LIN {X 0.085,Y -554.089,Z 631.442,A 0.000,B 0.000,C 90.000,E1 115.540} C_DIS
LIN {X 0.039,Y -558.217,Z 631.438,A 0.000,B 0.000,C 90.000,E1 114.847} C_DIS
LIN {X 0.028,Y -561.886,Z 631.434,A 0.000,B 0.000,C 90.000,E1 114.155} C_DIS
LIN {X -0.047,Y -565.879,Z 631.430,A 0.000,B 0.000,C 90.000,E1 113.334} C_DIS
LIN {X 0.254,Y -570.586,Z 631.424,A 0.000,B 0.000,C 90.000,E1 112.206} C_DIS
LIN {X 0.040,Y -573.804,Z 631.419,A 0.000,B 0.000,C 90.000,E1 111.408} C_DIS
LIN {X 0.026,Y -575.811,Z 631.416,A 0.000,B 0.000,C 90.000,E1 110.865} C_DIS
LIN {X -0.133,Y -578.606,Z 631.411,A 0.000,B 0.000,C 90.000,E1 110.066} C_DIS
LIN {X -0.267,Y -581.153,Z 631.407,A 0.000,B 0.000,C 90.000,E1 109.268} C_DIS
LIN {X 0.171,Y -583.428,Z 631.402,A 0.000,B 0.000,C 90.000,E1 108.417} C_DIS
LIN {X -0.105,Y -585.449,Z 631.398,A 0.000,B 0.000,C 90.000,E1 107.638} C_DIS
LIN {X 0.203,Y -587.394,Z 631.393,A 0.000,B 0.000,C 90.000,E1 106.804} C_DIS
LIN {X 0.014,Y -591.886,Z 631.383,A 0.000,B 0.000,C 90.000,E1 104.954} C_DIS
LIN {X 0.067,Y -595.897,Z 631.374,A 0.000,B 0.000,C 90.000,E1 103.355} C_DIS
LIN {X -0.234,Y -599.246,Z 631.367,A 0.000,B 0.000,C 90.000,E1 102.063} C_DIS
LIN {X 0.103,Y -602.617,Z 631.360,A 0.000,B 0.000,C 90.000,E1 100.715} C_DIS
LIN {X -0.213,Y -605.836,Z 631.352,A 0.000,B 0.000,C 90.000,E1 99.434} C_DIS
LIN {X 0.029,Y -608.811,Z 631.345,A 0.000,B 0.000,C 90.000,E1 98.106} C_DIS
LIN {X -0.005,Y -611.109,Z 631.339,A 0.000,B 0.000,C 90.000,E1 97.068} C_DIS
LIN {X -0.273,Y -613.680,Z 631.332,A 0.000,B 0.000,C 90.000,E1 95.796} C_DIS
LIN {X 0.024,Y -615.053,Z 631.328,A 0.000,B 0.000,C 90.000,E1 94.992} C_DIS
LIN {X -0.248,Y -617.171,Z 631.321,A 0.000,B 0.000,C 90.000,E1 93.726} C_DIS
LIN {X -0.222,Y -618.720,Z 631.315,A 0.000,B 0.000,C 90.000,E1 92.694} C_DIS
LIN {X 0.139,Y -620.287,Z 631.308,A 0.000,B 0.000,C 90.000,E1 91.375} C_DIS
LIN {X -0.136,Y -621.077,Z 631.303,A 0.000,B 0.000,C 90.000,E1 90.630} C_DIS
LIN {X -0.075,Y -621.849,Z 631.298,A 0.000,B 0.000,C 90.000,E1 89.599} C_DIS
LIN {X -0.301,Y -622.416,Z 631.291,A 0.000,B 0.000,C 90.000,E1 88.339} C_DIS
LIN {X -0.208,Y -622.576,Z 631.285,A 0.000,B 0.000,C 90.000,E1 87.306} C_DIS
LIN {X 0.211,Y -622.380,Z 631.278,A 0.000,B 0.000,C 90.000,E1 85.988} C_DIS
LIN {X -0.270,Y -621.941,Z 631.272,A 0.000,B 0.000,C 90.000,E1 85.008} C_DIS
LIN {X 0.183,Y -621.213,Z 631.265,A 0.000,B 0.000,C 90.000,E1 83.685} C_DIS
LIN {X 0.073,Y -620.135,Z 631.258,A 0.000,B 0.000,C 90.000,E1 82.413} C_DIS
LIN {X -0.104,Y -619.289,Z 631.254,A 0.000,B 0.000,C 90.000,E1 81.659} C_DIS
LIN {X -0.012,Y -617.891,Z 631.248,A 0.000,B 0.000,C 90.000,E1 80.622} C_DIS
LIN {X 0.151,Y -616.382,Z 631.242,A 0.000,B 0.000,C 90.000,E1 79.577} C_DIS
LIN {X 0.168,Y -614.185,Z 631.235,A 0.000,B 0.000,C 90.000,E1 78.285} C_DIS
LIN {X -0.194,Y -612.299,Z 631.229,A 0.000,B 0.000,C 90.000,E1 77.285} C_DIS
LIN {X -0.233,Y -609.621,Z 631.222,A 0.000,B 0.000,C 90.000,E1 75.992} C_DIS
LIN {X -0.071,Y -607.405,Z 631.216,A 0.000,B 0.000,C 90.000,E1 74.936} C_DIS
LIN {X 0.112,Y -604.394,Z 631.209,A 0.000,B 0.000,C 90.000,E1 73.614} C_DIS
LIN {X -0.222,Y -601.806,Z 631.203,A 0.000,B 0.000,C 90.000,E1 72.598} C_DIS
LIN {X 0.262,Y -599.743,Z 631.199,A 0.000,B 0.000,C 90.000,E1 71.764} C_DIS
LIN {X -0.126,Y -598.233,Z 631.196,A 0.000,B 0.000,C 90.000,E1 71.275} C_DIS
LIN {X -0.057,Y -595.727,Z 631.192,A 0.000,B 0.000,C 90.000,E1 70.477} C_DIS
LIN {X 0.096,Y -594.011,Z 631.189,A 0.000,B 0.000,C 90.000,E1 69.934} C_DIS
LIN {X -0.197,Y -590.097,Z 631.183,A 0.000,B 0.000,C 90.000,E1 68.901} C_DIS
LIN {X -0.210,Y -586.932,Z 631.178,A 0.000,B 0.000,C 90.000,E1 68.103} C_DIS
LIN {X -0.034,Y -583.567,Z 631.174,A 0.000,B 0.000,C 90.000,E1 67.283} C_DIS
LIN {X -0.187,Y -579.320,Z 631.169,A 0.000,B 0.000,C 90.000,E1 66.357} C_DIS
LIN {X -0.091,Y -575.356,Z 631.164,A 0.000,B 0.000,C 90.000,E1 65.537} C_DIS
LIN {X 0.139,Y -572.004,Z 631.160,A 0.000,B 0.000,C 90.000,E1 64.845} C_DIS
LIN {X 0.152,Y -567.287,Z 631.156,A 0.000,B 0.000,C 90.000,E1 64.024} C_DIS
LIN {X -0.069,Y -564.081,Z 631.153,A 0.000,B 0.000,C 90.000,E1 63.512} C_DIS
LIN {X -0.045,Y -559.282,Z 631.149,A 0.000,B 0.000,C 90.000,E1 62.820} C_DIS
LIN {X -0.196,Y -555.143,Z 631.146,A 0.000,B 0.000,C 90.000,E1 62.281} C_DIS
LIN {X -0.143,Y -550.650,Z 631.143,A 0.000,B 0.000,C 90.000,E1 61.719} C_DIS
LIN {X -0.182,Y -545.605,Z 631.140,A 0.000,B 0.000,C 90.000,E1 61.179} C_DIS
LIN {X -0.231,Y -541.679,Z 631.138,A 0.000,B 0.000,C 90.000,E1 60.795} C_DIS
LIN {X -0.230,Y -536.321,Z 631.135,A 0.000,B 0.000,C 90.000,E1 60.333} C_DIS
LIN {X -0.030,Y -530.617,Z 631.133,A 0.000,B 0.000,C 90.000,E1 59.871} C_DIS
LIN {X -0.118,Y -524.164,Z 631.130,A 0.000,B 0.000,C 90.000,E1 59.459} C_DIS
LIN {X 0.119,Y -515.999,Z 631.128,A 0.000,B 0.000,C 90.000,E1 58.948} C_DIS
LIN {X 0.131,Y -510.785,Z 631.126,A 0.000,B 0.000,C 90.000,E1 58.663} C_DIS
LIN {X -0.016,Y -503.911,Z 631.124,A 0.000,B 0.000,C 90.000,E1 58.329} C_DIS
LIN {X -0.137,Y -488.724,Z 631.120,A 0.000,B 0.000,C 90.000,E1 57.582} C_DIS
LIN {X -0.265,Y -467.090,Z 631.114,A 0.000,B 0.000,C 90.000,E1 56.501} C_DIS
LIN {X 0.064,Y -445.248,Z 631.107,A 0.000,B 0.000,C 90.000,E1 55.308} C_DIS
LIN {X -0.003,Y -440.385,Z 631.106,A 0.000,B 0.000,C 90.000,E1 55.055} C_DIS
LIN {X -0.047,Y -440.315,Z 631.106,A 0.000,B 0.000,C 90.000,E1 55.055} C_DIS
LIN {X -0.113,Y -431.751,Z 631.083,A 0.000,B 0.000,C 90.000,E1 50.964} C_DIS
LIN {X 0.067,Y -430.164,Z 631.079,A 0.000,B 0.000,C 90.000,E1 50.275} C_DIS
LIN {X -0.052,Y -425.382,Z 631.068,A 0.000,B 0.000,C 90.000,E1 48.243} C_DIS
LIN {X -0.081,Y -425.960,Z 631.061,A 0.000,B 0.000,C 90.000,E1 46.944} C_DIS
LIN {X 0.079,Y -426.371,Z 631.051,A 0.000,B 0.000,C 90.000,E1 45.243} C_DIS
LIN {X -0.214,Y -427.010,Z 631.038,A 0.000,B 0.000,C 90.000,E1 42.933} C_DIS
LIN {X 0.135,Y -427.902,Z 631.025,A 0.000,B 0.000,C 90.000,E1 40.539} C_DIS
LIN {X -0.059,Y -428.921,Z 631.012,A 0.000,B 0.000,C 90.000,E1 38.222} C_DIS
LIN {X -0.065,Y -429.888,Z 631.001,A 0.000,B 0.000,C 90.000,E1 36.217} C_DIS
LIN {X 0.053,Y -430.598,Z 630.992,A 0.000,B 0.000,C 90.000,E1 34.532} C_DIS
LIN {X 0.054,Y -430.923,Z 630.988,A 0.000,B 0.000,C 90.000,E1 33.865} C_DIS
LIN {X -0.039,Y -431.638,Z 630.977,A 0.000,B 0.000,C 90.000,E1 31.878} C_DIS
LIN {X 0.030,Y -432.485,Z 630.964,A 0.000,B 0.000,C 90.000,E1 29.539} C_DIS
LIN {X 0.267,Y -433.344,Z 630.953,A 0.000,B 0.000,C 90.000,E1 27.513} C_DIS
LIN {X 0.133,Y -434.356,Z 630.940,A 0.000,B 0.000,C 90.000,E1 25.207} C_DIS
LIN {X 0.057,Y -435.441,Z 630.927,A 0.000,B 0.000,C 90.000,E1 22.898} C_DIS
LIN {X 0.182,Y -436.359,Z 630.918,A 0.000,B 0.000,C 90.000,E1 21.227} C_DIS
LIN {X -0.077,Y -437.108,Z 630.911,A 0.000,B 0.000,C 90.000,E1 19.939} C_DIS
LIN {X 0.026,Y -438.151,Z 630.900,A 0.000,B 0.000,C 90.000,E1 17.946} C_DIS
LIN {X 0.025,Y -439.291,Z 630.889,A 0.000,B 0.000,C 90.000,E1 15.969} C_DIS
LIN {X -0.100,Y -440.959,Z 630.874,A 0.000,B 0.000,C 90.000,E1 13.355} C_DIS
LIN {X -0.207,Y -442.712,Z 630.861,A 0.000,B 0.000,C 90.000,E1 11.074} C_DIS
LIN {X -0.175,Y -444.938,Z 630.847,A 0.000,B 0.000,C 90.000,E1 8.454} C_DIS
LIN {X -0.071,Y -446.894,Z 630.836,A 0.000,B 0.000,C 90.000,E1 6.486} C_DIS
LIN {X -0.151,Y -449.638,Z 630.822,A 0.000,B 0.000,C 90.000,E1 3.898} C_DIS
LIN {X 0.198,Y -451.560,Z 630.813,A 0.000,B 0.000,C 90.000,E1 2.236} C_DIS
LIN {X -0.106,Y -455.171,Z 630.797,A 0.000,B 0.000,C 90.000,E1 359.484} C_DIS
LIN {X -0.178,Y -458.582,Z 630.785,A 0.000,B 0.000,C 90.000,E1 357.249} C_DIS
LIN {X -0.107,Y -462.241,Z 630.772,A 0.000,B 0.000,C 90.000,E1 355.008} C_DIS
LIN {X 0.109,Y -466.017,Z 630.760,A 0.000,B 0.000,C 90.000,E1 352.761} C_DIS
LIN {X -0.192,Y -469.281,Z 630.749,A 0.000,B 0.000,C 90.000,E1 350.905} C_DIS
LIN {X -0.249,Y -471.967,Z 630.741,A 0.000,B 0.000,C 90.000,E1 349.342} C_DIS
LIN {X 0.053,Y -475.727,Z 630.729,A 0.000,B 0.000,C 90.000,E1 347.117} C_DIS
LIN {X 0.098,Y -479.596,Z 630.716,A 0.000,B 0.000,C 90.000,E1 344.936} C_DIS
LIN {X 0.040,Y -483.665,Z 630.704,A 0.000,B 0.000,C 90.000,E1 342.779} C_DIS
LIN {X -0.241,Y -486.681,Z 630.696,A 0.000,B 0.000,C 90.000,E1 341.275} C_DIS
LIN {X 0.149,Y -489.655,Z 630.687,A 0.000,B 0.000,C 90.000,E1 339.699} C_DIS
LIN {X -0.107,Y -493.167,Z 630.677,A 0.000,B 0.000,C 90.000,E1 337.901} C_DIS
LIN {X 0.025,Y -494.765,Z 630.672,A 0.000,B 0.000,C 90.000,E1 336.975} C_DIS
LIN {X -0.180,Y -497.255,Z 630.664,A 0.000,B 0.000,C 90.000,E1 335.485} C_DIS
LIN {X 0.076,Y -499.568,Z 630.655,A 0.000,B 0.000,C 90.000,E1 333.948} C_DIS
LIN {X 0.002,Y -502.293,Z 630.645,A 0.000,B 0.000,C 90.000,E1 332.153} C_DIS
LIN {X 0.149,Y -506.008,Z 630.632,A 0.000,B 0.000,C 90.000,E1 329.744} C_DIS
LIN {X 0.148,Y -509.819,Z 630.620,A 0.000,B 0.000,C 90.000,E1 327.661} C_DIS
LIN {X -0.162,Y -513.440,Z 630.612,A 0.000,B 0.000,C 90.000,E1 326.215} C_DIS
LIN {X 0.103,Y -515.315,Z 630.609,A 0.000,B 0.000,C 90.000,E1 325.595} C_DIS
LIN {X 0.028,Y -516.613,Z 630.607,A 0.000,B 0.000,C 90.000,E1 325.308} C_DIS
LIN {X -0.028,Y -518.300,Z 630.605,A 0.000,B 0.000,C 90.000,E1 324.975} C_DIS
LIN {X 0.088,Y -519.185,Z 630.605,A 0.000,B 0.000,C 90.000,E1 324.815} C_DIS
LIN {X -0.264,Y -520.383,Z 630.604,A 0.000,B 0.000,C 90.000,E1 324.689} C_DIS
LIN {X 0.103,Y -522.215,Z 630.602,A 0.000,B 0.000,C 90.000,E1 324.356} C_DIS
LIN {X -0.089,Y -526.231,Z 630.599,A 0.000,B 0.000,C 90.000,E1 323.909} C_DIS
LIN {X 0.108,Y -531.100,Z 630.597,A 0.000,B 0.000,C 90.000,E1 323.417} C_DIS
LIN {X -0.048,Y -534.048,Z 630.595,A 0.000,B 0.000,C 90.000,E1 323.176} C_DIS
LIN {X -0.132,Y -540.909,Z 630.592,A 0.000,B 0.000,C 90.000,E1 322.637} C_DIS
LIN {X -0.285,Y -550.938,Z 630.588,A 0.000,B 0.000,C 90.000,E1 321.823} C_DIS
LIN {X 0.137,Y -563.763,Z 630.582,A 0.000,B 0.000,C 90.000,E1 320.723} C_DIS
LIN {X -0.050,Y -572.217,Z 630.578,A 0.000,B 0.000,C 90.000,E1 320.033} C_DIS
LIN {X -0.220,Y -581.991,Z 630.573,A 0.000,B 0.000,C 90.000,E1 319.218} C_DIS
LIN {X -0.098,Y -590.110,Z 630.569,A 0.000,B 0.000,C 90.000,E1 318.485} C_DIS
LIN {X 0.000,Y -597.970,Z 630.565,A 0.000,B 0.000,C 90.000,E1 317.757} C_DIS
LIN {X -0.241,Y -602.878,Z 630.563,A 0.000,B 0.000,C 90.000,E1 317.310} C_DIS
LIN {X 0.060,Y -605.489,Z 630.561,A 0.000,B 0.000,C 90.000,E1 317.025} C_DIS
LIN {X 0.076,Y -610.159,Z 630.559,A 0.000,B 0.000,C 90.000,E1 316.539} C_DIS
LIN {X 0.043,Y -614.632,Z 630.556,A 0.000,B 0.000,C 90.000,E1 316.053} C_DIS
LIN {X -0.024,Y -618.922,Z 630.553,A 0.000,B 0.000,C 90.000,E1 315.567} C_DIS
LIN {X -0.329,Y -623.212,Z 630.550,A 0.000,B 0.000,C 90.000,E1 315.081} C_DIS
LIN {X -0.351,Y -630.233,Z 630.545,A 0.000,B 0.000,C 90.000,E1 314.190} C_DIS
LIN {X 0.165,Y -636.856,Z 630.540,A 0.000,B 0.000,C 90.000,E1 313.257} C_DIS
LIN {X 0.009,Y -642.290,Z 630.536,A 0.000,B 0.000,C 90.000,E1 312.528} C_DIS
LIN {X -0.239,Y -648.488,Z 630.531,A 0.000,B 0.000,C 90.000,E1 311.676} C_DIS
LIN {X 0.072,Y -654.390,Z 630.527,A 0.000,B 0.000,C 90.000,E1 310.782} C_DIS
LIN {X -0.005,Y -658.239,Z 630.523,A 0.000,B 0.000,C 90.000,E1 310.172} C_DIS
LIN {X -0.080,Y -661.081,Z 630.521,A 0.000,B 0.000,C 90.000,E1 309.688} C_DIS
LIN {X -0.018,Y -664.314,Z 630.517,A 0.000,B 0.000,C 90.000,E1 309.072} C_DIS
LIN {X -0.064,Y -666.726,Z 630.514,A 0.000,B 0.000,C 90.000,E1 308.588} C_DIS
LIN {X 0.093,Y -671.048,Z 630.509,A 0.000,B 0.000,C 90.000,E1 307.604} C_DIS
LIN {X 0.190,Y -673.983,Z 630.505,A 0.000,B 0.000,C 90.000,E1 306.870} C_DIS
LIN {X -0.088,Y -676.736,Z 630.501,A 0.000,B 0.000,C 90.000,E1 306.171} C_DIS
LIN {X 0.215,Y -680.835,Z 630.494,A 0.000,B 0.000,C 90.000,E1 304.945} C_DIS
LIN {X 0.181,Y -683.858,Z 630.489,A 0.000,B 0.000,C 90.000,E1 303.992} C_DIS
LIN {X -0.005,Y -686.037,Z 630.485,A 0.000,B 0.000,C 90.000,E1 303.293} C_DIS
LIN {X 0.246,Y -689.601,Z 630.478,A 0.000,B 0.000,C 90.000,E1 302.084} C_DIS
LIN {X 0.330,Y -692.272,Z 630.473,A 0.000,B 0.000,C 90.000,E1 301.131} C_DIS
LIN {X -0.267,Y -695.505,Z 630.467,A 0.000,B 0.000,C 90.000,E1 300.001} C_DIS
LIN {X 0.051,Y -698.955,Z 630.459,A 0.000,B 0.000,C 90.000,E1 298.565} C_DIS
LIN {X -0.111,Y -701.035,Z 630.454,A 0.000,B 0.000,C 90.000,E1 297.641} C_DIS
LIN {X 0.087,Y -702.418,Z 630.450,A 0.000,B 0.000,C 90.000,E1 296.924} C_DIS
LIN {X -0.018,Y -703.452,Z 630.446,A 0.000,B 0.000,C 90.000,E1 296.232} C_DIS
LIN {X -0.085,Y -703.687,Z 630.443,A 0.000,B 0.000,C 90.000,E1 295.771} C_DIS
LIN {X -0.107,Y -703.580,Z 630.442,A 0.000,B 0.000,C 90.000,E1 295.540} C_DIS
LIN {X -0.176,Y -702.515,Z 630.439,A 0.000,B 0.000,C 90.000,E1 295.079} C_DIS
LIN {X 0.104,Y -701.665,Z 630.438,A 0.000,B 0.000,C 90.000,E1 294.823} C_DIS
LIN {X 0.225,Y -699.045,Z 630.436,A 0.000,B 0.000,C 90.000,E1 294.463} C_DIS
LIN {X -0.143,Y -697.041,Z 630.435,A 0.000,B 0.000,C 90.000,E1 294.259} C_DIS
LIN {X -0.012,Y -695.571,Z 630.434,A 0.000,B 0.000,C 90.000,E1 294.131} C_DIS
LIN {X -0.023,Y -693.395,Z 630.434,A 0.000,B 0.000,C 90.000,E1 294.027} C_DIS
LIN {X 0.255,Y -686.989,Z 630.432,A 0.000,B 0.000,C 90.000,E1 293.770} C_DIS
LIN {X -0.216,Y -683.102,Z 630.432,A 0.000,B 0.000,C 90.000,E1 293.695} C_DIS
LIN {X -0.155,Y -680.635,Z 630.431,A 0.000,B 0.000,C 90.000,E1 293.643} C_DIS
LIN {X 0.228,Y -674.010,Z 630.431,A 0.000,B 0.000,C 90.000,E1 293.515} C_DIS
LIN {X -0.254,Y -664.941,Z 630.430,A 0.000,B 0.000,C 90.000,E1 293.462} C_DIS
LIN {X -0.082,Y -651.280,Z 630.429,A 0.000,B 0.000,C 90.000,E1 293.259} C_DIS
LIN {X -0.303,Y -639.642,Z 630.428,A 0.000,B 0.000,C 90.000,E1 293.078} C_DIS
LIN {X -0.087,Y -628.867,Z 630.427,A 0.000,B 0.000,C 90.000,E1 292.823} C_DIS
LIN {X -0.031,Y -615.450,Z 630.425,A 0.000,B 0.000,C 90.000,E1 292.461} C_DIS
LIN {X -0.061,Y -594.878,Z 630.421,A 0.000,B 0.000,C 90.000,E1 291.844} C_DIS
LIN {X -0.126,Y -579.185,Z 630.419,A 0.000,B 0.000,C 90.000,E1 291.354} C_DIS
LIN {X -0.041,Y -570.243,Z 630.417,A 0.000,B 0.000,C 90.000,E1 291.099} C_DIS
LIN {X -0.246,Y -563.976,Z 630.416,A 0.000,B 0.000,C 90.000,E1 290.918} C_DIS
LIN {X -0.301,Y -559.805,Z 630.415,A 0.000,B 0.000,C 90.000,E1 290.737} C_DIS
LIN {X 0.159,Y -558.684,Z 630.415,A 0.000,B 0.000,C 90.000,E1 290.610} C_DIS
LIN {X -0.035,Y -556.909,Z 630.414,A 0.000,B 0.000,C 90.000,E1 290.482} C_DIS
LIN {X -0.070,Y -556.884,Z 630.414,A 0.000,B 0.000,C 90.000,E1 290.482} C_DIS
LIN {X 0.037,Y -556.255,Z 630.413,A 0.000,B 0.000,C 90.000,E1 290.248} C_DIS
LIN {X 0.215,Y -555.883,Z 630.410,A 0.000,B 0.000,C 90.000,E1 289.812} C_DIS
LIN {X -0.241,Y -556.063,Z 630.406,A 0.000,B 0.000,C 90.000,E1 289.033} C_DIS
LIN {X -0.208,Y -556.015,Z 630.398,A 0.000,B 0.000,C 90.000,E1 287.638} C_DIS
LIN {X 0.063,Y -555.727,Z 630.392,A 0.000,B 0.000,C 90.000,E1 286.496} C_DIS
LIN {X 0.173,Y -555.389,Z 630.386,A 0.000,B 0.000,C 90.000,E1 285.371} C_DIS
LIN {X -0.130,Y -554.702,Z 630.378,A 0.000,B 0.000,C 90.000,E1 284.008} C_DIS
LIN {X 0.216,Y -553.824,Z 630.369,A 0.000,B 0.000,C 90.000,E1 282.299} C_DIS
LIN {X -0.246,Y -553.157,Z 630.361,A 0.000,B 0.000,C 90.000,E1 280.950} C_DIS
LIN {X -0.162,Y -552.433,Z 630.351,A 0.000,B 0.000,C 90.000,E1 279.265} C_DIS
LIN {X -0.174,Y -551.722,Z 630.342,A 0.000,B 0.000,C 90.000,E1 277.587} C_DIS
LIN {X -0.161,Y -550.947,Z 630.331,A 0.000,B 0.000,C 90.000,E1 275.625} C_DIS
LIN {X -0.223,Y -550.382,Z 630.320,A 0.000,B 0.000,C 90.000,E1 273.669} C_DIS
LIN {X 0.130,Y -549.922,Z 630.311,A 0.000,B 0.000,C 90.000,E1 271.949} C_DIS
LIN {X -0.130,Y -549.551,Z 630.303,A 0.000,B 0.000,C 90.000,E1 270.573} C_DIS
LIN {X 0.087,Y -549.082,Z 630.297,A 0.000,B 0.000,C 90.000,E1 269.427} C_DIS
LIN {X -0.189,Y -548.444,Z 630.289,A 0.000,B 0.000,C 90.000,E1 268.051} C_DIS
LIN {X 0.076,Y -547.871,Z 630.281,A 0.000,B 0.000,C 90.000,E1 266.617} C_DIS
LIN {X -0.228,Y -547.096,Z 630.273,A 0.000,B 0.000,C 90.000,E1 265.241} C_DIS
LIN {X 0.199,Y -545.764,Z 630.263,A 0.000,B 0.000,C 90.000,E1 263.223} C_DIS
LIN {X -0.147,Y -545.026,Z 630.258,A 0.000,B 0.000,C 90.000,E1 262.413} C_DIS
LIN {X 0.127,Y -543.834,Z 630.252,A 0.000,B 0.000,C 90.000,E1 261.254} C_DIS
LIN {X 0.075,Y -541.448,Z 630.239,A 0.000,B 0.000,C 90.000,E1 258.993} C_DIS
LIN {X 0.001,Y -539.980,Z 630.229,A 0.000,B 0.000,C 90.000,E1 257.297} C_DIS
LIN {X 0.012,Y -538.583,Z 630.220,A 0.000,B 0.000,C 90.000,E1 255.589} C_DIS
LIN {X 0.016,Y -537.544,Z 630.214,A 0.000,B 0.000,C 90.000,E1 254.448} C_DIS
LIN {X 0.115,Y -535.708,Z 630.204,A 0.000,B 0.000,C 90.000,E1 252.725} C_DIS
LIN {X -0.189,Y -534.014,Z 630.195,A 0.000,B 0.000,C 90.000,E1 251.040} C_DIS
LIN {X -0.269,Y -533.017,Z 630.190,A 0.000,B 0.000,C 90.000,E1 250.188} C_DIS
LIN {X -0.164,Y -531.434,Z 630.183,A 0.000,B 0.000,C 90.000,E1 249.028} C_DIS
LIN {X 0.111,Y -529.754,Z 630.177,A 0.000,B 0.000,C 90.000,E1 247.847} C_DIS
LIN {X -0.121,Y -527.856,Z 630.171,A 0.000,B 0.000,C 90.000,E1 246.719} C_DIS
LIN {X 0.105,Y -525.750,Z 630.164,A 0.000,B 0.000,C 90.000,E1 245.537} C_DIS
LIN {X 0.127,Y -524.095,Z 630.159,A 0.000,B 0.000,C 90.000,E1 244.665} C_DIS
LIN {X 0.180,Y -520.981,Z 630.151,A 0.000,B 0.000,C 90.000,E1 243.204} C_DIS
LIN {X 0.071,Y -517.162,Z 630.142,A 0.000,B 0.000,C 90.000,E1 241.463} C_DIS
LIN {X 0.115,Y -514.546,Z 630.135,A 0.000,B 0.000,C 90.000,E1 240.284} C_DIS
LIN {X 0.030,Y -512.489,Z 630.130,A 0.000,B 0.000,C 90.000,E1 239.410} C_DIS
LIN {X 0.170,Y -508.945,Z 630.122,A 0.000,B 0.000,C 90.000,E1 237.916} C_DIS
LIN {X 0.246,Y -505.244,Z 630.114,A 0.000,B 0.000,C 90.000,E1 236.421} C_DIS
LIN {X -0.056,Y -502.256,Z 630.107,A 0.000,B 0.000,C 90.000,E1 235.261} C_DIS
LIN {X -0.118,Y -499.092,Z 630.100,A 0.000,B 0.000,C 90.000,E1 234.069} C_DIS
LIN {X 0.056,Y -492.078,Z 630.085,A 0.000,B 0.000,C 90.000,E1 231.331} C_DIS
LIN {X -0.098,Y -488.282,Z 630.077,A 0.000,B 0.000,C 90.000,E1 229.828} C_DIS
LIN {X 0.004,Y -484.582,Z 630.068,A 0.000,B 0.000,C 90.000,E1 228.286} C_DIS
LIN {X -0.162,Y -480.044,Z 630.058,A 0.000,B 0.000,C 90.000,E1 226.458} C_DIS
LIN {X -0.018,Y -474.760,Z 630.046,A 0.000,B 0.000,C 90.000,E1 224.271} C_DIS
LIN {X 0.235,Y -470.463,Z 630.036,A 0.000,B 0.000,C 90.000,E1 222.366} C_DIS
LIN {X -0.005,Y -467.058,Z 630.027,A 0.000,B 0.000,C 90.000,E1 220.825} C_DIS
LIN {X -0.254,Y -463.651,Z 630.018,A 0.000,B 0.000,C 90.000,E1 219.277} C_DIS
LIN {X -0.171,Y -459.645,Z 630.008,A 0.000,B 0.000,C 90.000,E1 217.363} C_DIS
LIN {X 0.000,Y -455.235,Z 629.995,A 0.000,B 0.000,C 90.000,E1 215.105} C_DIS
LIN {X 0.081,Y -451.710,Z 629.984,A 0.000,B 0.000,C 90.000,E1 213.166} C_DIS
LIN {X -0.093,Y -447.591,Z 629.972,A 0.000,B 0.000,C 90.000,E1 210.924} C_DIS
LIN {X 0.096,Y -444.173,Z 629.961,A 0.000,B 0.000,C 90.000,E1 208.949} C_DIS
LIN {X -0.009,Y -440.665,Z 629.950,A 0.000,B 0.000,C 90.000,E1 207.001} C_DIS
LIN {X 0.137,Y -438.382,Z 629.943,A 0.000,B 0.000,C 90.000,E1 205.668} C_DIS
LIN {X 0.084,Y -434.772,Z 629.932,A 0.000,B 0.000,C 90.000,E1 203.695} C_DIS
LIN {X 0.175,Y -431.877,Z 629.923,A 0.000,B 0.000,C 90.000,E1 202.025} C_DIS
LIN {X 0.075,Y -427.901,Z 629.910,A 0.000,B 0.000,C 90.000,E1 199.704} C_DIS
LIN {X 0.135,Y -424.096,Z 629.897,A 0.000,B 0.000,C 90.000,E1 197.347} C_DIS
LIN {X 0.126,Y -421.492,Z 629.887,A 0.000,B 0.000,C 90.000,E1 195.662} C_DIS
LIN {X -0.165,Y -418.953,Z 629.878,A 0.000,B 0.000,C 90.000,E1 194.008} C_DIS
LIN {X -0.042,Y -415.754,Z 629.866,A 0.000,B 0.000,C 90.000,E1 191.951} C_DIS
LIN {X -0.005,Y -411.834,Z 629.851,A 0.000,B 0.000,C 90.000,E1 189.208} C_DIS
LIN {X 0.101,Y -409.424,Z 629.842,A 0.000,B 0.000,C 90.000,E1 187.473} C_DIS
LIN {X 0.142,Y -405.681,Z 629.826,A 0.000,B 0.000,C 90.000,E1 184.702} C_DIS
LIN {X -0.067,Y -402.437,Z 629.811,A 0.000,B 0.000,C 90.000,E1 181.949} C_DIS
LIN {X -0.026,Y -399.449,Z 629.793,A 0.000,B 0.000,C 90.000,E1 178.797} C_DIS
LIN {X 0.144,Y -396.808,Z 629.768,A 0.000,B 0.000,C 90.000,E1 174.204} C_DIS
LIN {X -0.189,Y -396.039,Z 629.752,A 0.000,B 0.000,C 90.000,E1 171.432} C_DIS
LIN {X 0.064,Y -395.686,Z 629.739,A 0.000,B 0.000,C 90.000,E1 168.926} C_DIS
LIN {X -0.032,Y -395.779,Z 629.723,A 0.000,B 0.000,C 90.000,E1 166.117} C_DIS
LIN {X 0.131,Y -396.029,Z 629.711,A 0.000,B 0.000,C 90.000,E1 163.976} C_DIS
LIN {X 0.107,Y -396.478,Z 629.697,A 0.000,B 0.000,C 90.000,E1 161.511} C_DIS
LIN {X -0.155,Y -397.099,Z 629.684,A 0.000,B 0.000,C 90.000,E1 159.082} C_DIS
LIN {X 0.096,Y -397.908,Z 629.668,A 0.000,B 0.000,C 90.000,E1 156.230} C_DIS
LIN {X -0.128,Y -398.490,Z 629.656,A 0.000,B 0.000,C 90.000,E1 154.152} C_DIS
LIN {X 0.133,Y -399.066,Z 629.647,A 0.000,B 0.000,C 90.000,E1 152.359} C_DIS
LIN {X 0.122,Y -399.672,Z 629.635,A 0.000,B 0.000,C 90.000,E1 150.255} C_DIS
LIN {X 0.217,Y -400.386,Z 629.621,A 0.000,B 0.000,C 90.000,E1 147.788} C_DIS
LIN {X -0.023,Y -401.048,Z 629.610,A 0.000,B 0.000,C 90.000,E1 145.722} C_DIS
LIN {X 0.103,Y -402.033,Z 629.596,A 0.000,B 0.000,C 90.000,E1 143.256} C_DIS
LIN {X -0.084,Y -402.722,Z 629.586,A 0.000,B 0.000,C 90.000,E1 141.537} C_DIS
LIN {X -0.019,Y -403.341,Z 629.577,A 0.000,B 0.000,C 90.000,E1 139.784} C_DIS
LIN {X -0.168,Y -404.042,Z 629.565,A 0.000,B 0.000,C 90.000,E1 137.715} C_DIS
LIN {X -0.153,Y -404.538,Z 629.555,A 0.000,B 0.000,C 90.000,E1 135.972} C_DIS
LIN {X 0.159,Y -405.111,Z 629.546,A 0.000,B 0.000,C 90.000,E1 134.190} C_DIS
LIN {X -0.001,Y -406.211,Z 629.530,A 0.000,B 0.000,C 90.000,E1 131.434} C_DIS
LIN {X -0.177,Y -407.223,Z 629.521,A 0.000,B 0.000,C 90.000,E1 129.725} C_DIS
LIN {X -0.054,Y -408.248,Z 629.515,A 0.000,B 0.000,C 90.000,E1 128.669} C_DIS
LIN {X 0.094,Y -408.774,Z 629.513,A 0.000,B 0.000,C 90.000,E1 128.302} C_DIS
LIN {X -0.109,Y -412.610,Z 629.505,A 0.000,B 0.000,C 90.000,E1 126.950} C_DIS
LIN {X 0.099,Y -413.707,Z 629.504,A 0.000,B 0.000,C 90.000,E1 126.664} C_DIS
LIN {X 0.057,Y -414.262,Z 629.503,A 0.000,B 0.000,C 90.000,E1 126.583} C_DIS
LIN {X -0.213,Y -416.553,Z 629.502,A 0.000,B 0.000,C 90.000,E1 126.377} C_DIS
LIN {X -0.011,Y -420.672,Z 629.500,A 0.000,B 0.000,C 90.000,E1 126.011} C_DIS
LIN {X 0.055,Y -426.032,Z 629.498,A 0.000,B 0.000,C 90.000,E1 125.644} C_DIS
LIN {X -0.027,Y -446.098,Z 629.492,A 0.000,B 0.000,C 90.000,E1 124.485} C_DIS
LIN {X 0.034,Y -454.440,Z 629.489,A 0.000,B 0.000,C 90.000,E1 123.992} C_DIS
LIN {X -0.019,Y -462.488,Z 629.486,A 0.000,B 0.000,C 90.000,E1 123.499} C_DIS
LIN {X 0.096,Y -473.725,Z 629.482,A 0.000,B 0.000,C 90.000,E1 122.752} C_DIS
LIN {X -0.018,Y -480.082,Z 629.480,A 0.000,B 0.000,C 90.000,E1 122.339} C_DIS
LIN {X 0.171,Y -486.307,Z 629.477,A 0.000,B 0.000,C 90.000,E1 121.878} C_DIS
LIN {X -0.099,Y -494.021,Z 629.474,A 0.000,B 0.000,C 90.000,E1 121.337} C_DIS
LIN {X -0.026,Y -501.564,Z 629.471,A 0.000,B 0.000,C 90.000,E1 120.747} C_DIS
LIN {X 0.082,Y -507.495,Z 629.468,A 0.000,B 0.000,C 90.000,E1 120.256} C_DIS
LIN {X -0.133,Y -516.240,Z 629.464,A 0.000,B 0.000,C 90.000,E1 119.539} C_DIS
LIN {X -0.310,Y -523.189,Z 629.461,A 0.000,B 0.000,C 90.000,E1 118.949} C_DIS
LIN {X -0.048,Y -530.140,Z 629.457,A 0.000,B 0.000,C 90.000,E1 118.281} C_DIS
LIN {X -0.205,Y -535.464,Z 629.454,A 0.000,B 0.000,C 90.000,E1 117.769} C_DIS
LIN {X 0.012,Y -539.469,Z 629.452,A 0.000,B 0.000,C 90.000,E1 117.334} C_DIS
LIN {X -0.006,Y -545.258,Z 629.448,A 0.000,B 0.000,C 90.000,E1 116.668} C_DIS
LIN {X -0.140,Y -549.427,Z 629.445,A 0.000,B 0.000,C 90.000,E1 116.155} C_DIS
LIN {X -0.006,Y -552.319,Z 629.443,A 0.000,B 0.000,C 90.000,E1 115.720} C_DIS
LIN {X -0.124,Y -553.355,Z 629.442,A 0.000,B 0.000,C 90.000,E1 115.591} C_DIS
LIN {X 0.051,Y -557.531,Z 629.438,A 0.000,B 0.000,C 90.000,E1 114.899} C_DIS
LIN {X 0.074,Y -561.958,Z 629.434,A 0.000,B 0.000,C 90.000,E1 114.079} C_DIS
LIN {X 0.092,Y -565.424,Z 629.430,A 0.000,B 0.000,C 90.000,E1 113.387} C_DIS
LIN {X -0.174,Y -569.046,Z 629.425,A 0.000,B 0.000,C 90.000,E1 112.589} C_DIS
LIN {X -0.189,Y -572.439,Z 629.421,A 0.000,B 0.000,C 90.000,E1 111.770} C_DIS
LIN {X 0.148,Y -575.598,Z 629.416,A 0.000,B 0.000,C 90.000,E1 110.918} C_DIS
LIN {X -0.015,Y -578.472,Z 629.412,A 0.000,B 0.000,C 90.000,E1 110.120} C_DIS
LIN {X -0.152,Y -581.095,Z 629.407,A 0.000,B 0.000,C 90.000,E1 109.322} C_DIS
LIN {X 0.098,Y -583.447,Z 629.403,A 0.000,B 0.000,C 90.000,E1 108.489} C_DIS
LIN {X 0.232,Y -586.240,Z 629.397,A 0.000,B 0.000,C 90.000,E1 107.402} C_DIS
LIN {X 0.017,Y -590.738,Z 629.386,A 0.000,B 0.000,C 90.000,E1 105.552} C_DIS
LIN {X 0.175,Y -596.090,Z 629.375,A 0.000,B 0.000,C 90.000,E1 103.411} C_DIS
LIN {X 0.173,Y -600.172,Z 629.366,A 0.000,B 0.000,C 90.000,E1 101.827} C_DIS
LIN {X 0.101,Y -602.914,Z 629.360,A 0.000,B 0.000,C 90.000,E1 100.782} C_DIS
LIN {X -0.199,Y -606.199,Z 629.353,A 0.000,B 0.000,C 90.000,E1 99.500} C_DIS
LIN {X 0.148,Y -609.224,Z 629.345,A 0.000,B 0.000,C 90.000,E1 98.163} C_DIS
LIN {X -0.150,Y -612.122,Z 629.338,A 0.000,B 0.000,C 90.000,E1 96.891} C_DIS
LIN {X 0.140,Y -614.687,Z 629.331,A 0.000,B 0.000,C 90.000,E1 95.568} C_DIS
LIN {X 0.160,Y -615.590,Z 629.328,A 0.000,B 0.000,C 90.000,E1 95.049} C_DIS
LIN {X -0.103,Y -617.733,Z 629.321,A 0.000,B 0.000,C 90.000,E1 93.784} C_DIS
LIN {X -0.071,Y -619.314,Z 629.315,A 0.000,B 0.000,C 90.000,E1 92.751} C_DIS
LIN {X 0.261,Y -620.305,Z 629.311,A 0.000,B 0.000,C 90.000,E1 91.949} C_DIS
LIN {X -0.294,Y -621.472,Z 629.305,A 0.000,B 0.000,C 90.000,E1 90.974} C_DIS
LIN {X 0.065,Y -622.172,Z 629.301,A 0.000,B 0.000,C 90.000,E1 90.172} C_DIS
LIN {X -0.189,Y -622.693,Z 629.297,A 0.000,B 0.000,C 90.000,E1 89.427} C_DIS
LIN {X -0.111,Y -623.155,Z 629.291,A 0.000,B 0.000,C 90.000,E1 88.396} C_DIS
LIN {X -0.009,Y -623.281,Z 629.285,A 0.000,B 0.000,C 90.000,E1 87.364} C_DIS
LIN {X -0.196,Y -623.128,Z 629.278,A 0.000,B 0.000,C 90.000,E1 86.102} C_DIS
LIN {X -0.046,Y -622.656,Z 629.273,A 0.000,B 0.000,C 90.000,E1 85.065} C_DIS
LIN {X -0.198,Y -621.926,Z 629.266,A 0.000,B 0.000,C 90.000,E1 83.799} C_DIS
LIN {X 0.324,Y -620.828,Z 629.258,A 0.000,B 0.000,C 90.000,E1 82.470} C_DIS
LIN {X 0.065,Y -619.998,Z 629.254,A 0.000,B 0.000,C 90.000,E1 81.724} C_DIS
LIN {X 0.258,Y -618.589,Z 629.248,A 0.000,B 0.000,C 90.000,E1 80.679} C_DIS
LIN {X 0.196,Y -616.606,Z 629.241,A 0.000,B 0.000,C 90.000,E1 79.398} C_DIS
LIN {X 0.096,Y -614.344,Z 629.234,A 0.000,B 0.000,C 90.000,E1 78.117} C_DIS
LIN {X -0.270,Y -612.376,Z 629.228,A 0.000,B 0.000,C 90.000,E1 77.117} C_DIS
LIN {X -0.067,Y -610.190,Z 629.223,A 0.000,B 0.000,C 90.000,E1 76.061} C_DIS
LIN {X 0.253,Y -607.943,Z 629.217,A 0.000,B 0.000,C 90.000,E1 74.991} C_DIS
LIN {X -0.304,Y -604.898,Z 629.210,A 0.000,B 0.000,C 90.000,E1 73.740} C_DIS
LIN {X -0.058,Y -602.303,Z 629.204,A 0.000,B 0.000,C 90.000,E1 72.670} C_DIS
LIN {X 0.041,Y -600.186,Z 629.199,A 0.000,B 0.000,C 90.000,E1 71.873} C_DIS
LIN {X 0.227,Y -598.679,Z 629.196,A 0.000,B 0.000,C 90.000,E1 71.329} C_DIS
LIN {X 0.002,Y -595.235,Z 629.191,A 0.000,B 0.000,C 90.000,E1 70.296} C_DIS
LIN {X 0.151,Y -593.394,Z 629.188,A 0.000,B 0.000,C 90.000,E1 69.752} C_DIS
LIN {X 0.172,Y -590.380,Z 629.183,A 0.000,B 0.000,C 90.000,E1 68.954} C_DIS
LIN {X 0.163,Y -587.160,Z 629.179,A 0.000,B 0.000,C 90.000,E1 68.156} C_DIS
LIN {X 0.116,Y -583.747,Z 629.174,A 0.000,B 0.000,C 90.000,E1 67.358} C_DIS
LIN {X -0.042,Y -579.451,Z 629.169,A 0.000,B 0.000,C 90.000,E1 66.433} C_DIS
LIN {X 0.051,Y -575.453,Z 629.165,A 0.000,B 0.000,C 90.000,E1 65.613} C_DIS
LIN {X -0.253,Y -571.991,Z 629.161,A 0.000,B 0.000,C 90.000,E1 64.973} C_DIS
LIN {X -0.149,Y -568.043,Z 629.157,A 0.000,B 0.000,C 90.000,E1 64.280} C_DIS
LIN {X 0.098,Y -565.424,Z 629.155,A 0.000,B 0.000,C 90.000,E1 63.845} C_DIS
LIN {X -0.086,Y -563.770,Z 629.153,A 0.000,B 0.000,C 90.000,E1 63.589} C_DIS
LIN {X 0.277,Y -558.924,Z 629.149,A 0.000,B 0.000,C 90.000,E1 62.871} C_DIS
LIN {X 0.196,Y -554.991,Z 629.147,A 0.000,B 0.000,C 90.000,E1 62.359} C_DIS
LIN {X -0.125,Y -550.529,Z 629.144,A 0.000,B 0.000,C 90.000,E1 61.847} C_DIS
LIN {X -0.210,Y -545.398,Z 629.141,A 0.000,B 0.000,C 90.000,E1 61.307} C_DIS
LIN {X -0.302,Y -539.836,Z 629.138,A 0.000,B 0.000,C 90.000,E1 60.795} C_DIS
LIN {X 0.104,Y -535.373,Z 629.136,A 0.000,B 0.000,C 90.000,E1 60.383} C_DIS
LIN {X 0.077,Y -529.078,Z 629.133,A 0.000,B 0.000,C 90.000,E1 59.921} C_DIS
LIN {X -0.233,Y -522.296,Z 629.131,A 0.000,B 0.000,C 90.000,E1 59.537} C_DIS
LIN {X 0.012,Y -515.666,Z 629.129,A 0.000,B 0.000,C 90.000,E1 59.125} C_DIS
LIN {X -0.174,Y -510.596,Z 629.127,A 0.000,B 0.000,C 90.000,E1 58.869} C_DIS
LIN {X -0.290,Y -503.668,Z 629.125,A 0.000,B 0.000,C 90.000,E1 58.535} C_DIS
LIN {X -0.030,Y -485.162,Z 629.120,A 0.000,B 0.000,C 90.000,E1 57.582} C_DIS
LIN {X 0.129,Y -461.695,Z 629.113,A 0.000,B 0.000,C 90.000,E1 56.373} C_DIS
LIN {X 0.127,Y -443.131,Z 629.108,A 0.000,B 0.000,C 90.000,E1 55.388} C_DIS
LIN {X -0.173,Y -440.944,Z 629.107,A 0.000,B 0.000,C 90.000,E1 55.308} C_DIS
LIN {X 0.146,Y -440.878,Z 629.107,A 0.000,B 0.000,C 90.000,E1 55.261} C_DIS
LIN {X 0.025,Y -432.153,Z 629.084,A 0.000,B 0.000,C 90.000,E1 51.170} C_DIS
LIN {X -0.050,Y -431.559,Z 629.083,A 0.000,B 0.000,C 90.000,E1 50.848} C_DIS
LIN {X -0.174,Y -425.812,Z 629.069,A 0.000,B 0.000,C 90.000,E1 48.485} C_DIS
LIN {X 0.004,Y -426.517,Z 629.060,A 0.000,B 0.000,C 90.000,E1 46.824} C_DIS
LIN {X -0.032,Y -426.869,Z 629.053,A 0.000,B 0.000,C 90.000,E1 45.486} C_DIS
LIN {X 0.067,Y -427.415,Z 629.042,A 0.000,B 0.000,C 90.000,E1 43.461} C_DIS
LIN {X -0.095,Y -428.150,Z 629.030,A 0.000,B 0.000,C 90.000,E1 41.472} C_DIS
LIN {X -0.151,Y -428.851,Z 629.021,A 0.000,B 0.000,C 90.000,E1 39.806} C_DIS
LIN {X -0.225,Y -429.801,Z 629.010,A 0.000,B 0.000,C 90.000,E1 37.810} C_DIS
LIN {X -0.205,Y -430.731,Z 628.999,A 0.000,B 0.000,C 90.000,E1 35.804} C_DIS
LIN {X -0.065,Y -431.551,Z 628.988,A 0.000,B 0.000,C 90.000,E1 33.785} C_DIS
LIN {X -0.157,Y -432.147,Z 628.978,A 0.000,B 0.000,C 90.000,E1 32.133} C_DIS
LIN {X -0.079,Y -432.953,Z 628.966,A 0.000,B 0.000,C 90.000,E1 29.795} C_DIS
LIN {X 0.166,Y -433.772,Z 628.954,A 0.000,B 0.000,C 90.000,E1 27.769} C_DIS
LIN {X 0.045,Y -434.757,Z 628.942,A 0.000,B 0.000,C 90.000,E1 25.463} C_DIS
LIN {X -0.020,Y -435.770,Z 628.929,A 0.000,B 0.000,C 90.000,E1 23.153} C_DIS
LIN {X 0.108,Y -436.802,Z 628.918,A 0.000,B 0.000,C 90.000,E1 21.153} C_DIS
LIN {X 0.260,Y -437.520,Z 628.910,A 0.000,B 0.000,C 90.000,E1 19.812} C_DIS
LIN {X -0.047,Y -438.539,Z 628.899,A 0.000,B 0.000,C 90.000,E1 17.873} C_DIS
LIN {X -0.049,Y -439.668,Z 628.888,A 0.000,B 0.000,C 90.000,E1 15.898} C_DIS
LIN {X 0.001,Y -441.095,Z 628.876,A 0.000,B 0.000,C 90.000,E1 13.592} C_DIS
LIN {X -0.015,Y -442.804,Z 628.863,A 0.000,B 0.000,C 90.000,E1 11.299} C_DIS
LIN {X 0.007,Y -444.947,Z 628.848,A 0.000,B 0.000,C 90.000,E1 8.681} C_DIS
LIN {X 0.229,Y -447.194,Z 628.836,A 0.000,B 0.000,C 90.000,E1 6.372} C_DIS
LIN {X 0.165,Y -449.927,Z 628.821,A 0.000,B 0.000,C 90.000,E1 3.784} C_DIS
LIN {X 0.070,Y -451.812,Z 628.812,A 0.000,B 0.000,C 90.000,E1 2.178} C_DIS
LIN {X -0.104,Y -455.321,Z 628.797,A 0.000,B 0.000,C 90.000,E1 359.484} C_DIS
LIN {X 0.097,Y -458.214,Z 628.786,A 0.000,B 0.000,C 90.000,E1 357.535} C_DIS
LIN {X 0.125,Y -461.816,Z 628.774,A 0.000,B 0.000,C 90.000,E1 355.298} C_DIS
LIN {X -0.139,Y -465.570,Z 628.762,A 0.000,B 0.000,C 90.000,E1 353.109} C_DIS
LIN {X 0.009,Y -468.820,Z 628.751,A 0.000,B 0.000,C 90.000,E1 351.197} C_DIS
LIN {X -0.056,Y -471.496,Z 628.742,A 0.000,B 0.000,C 90.000,E1 349.634} C_DIS
LIN {X 0.234,Y -475.239,Z 628.730,A 0.000,B 0.000,C 90.000,E1 347.409} C_DIS
LIN {X -0.191,Y -479.067,Z 628.718,A 0.000,B 0.000,C 90.000,E1 345.283} C_DIS
LIN {X 0.067,Y -483.108,Z 628.706,A 0.000,B 0.000,C 90.000,E1 343.087} C_DIS
LIN {X -0.219,Y -486.746,Z 628.696,A 0.000,B 0.000,C 90.000,E1 341.275} C_DIS
LIN {X 0.198,Y -490.279,Z 628.686,A 0.000,B 0.000,C 90.000,E1 339.390} C_DIS
LIN {X -0.085,Y -493.196,Z 628.677,A 0.000,B 0.000,C 90.000,E1 337.901} C_DIS
LIN {X 0.048,Y -494.794,Z 628.672,A 0.000,B 0.000,C 90.000,E1 336.975} C_DIS
LIN {X -0.155,Y -497.282,Z 628.664,A 0.000,B 0.000,C 90.000,E1 335.485} C_DIS
LIN {X 0.101,Y -499.596,Z 628.655,A 0.000,B 0.000,C 90.000,E1 333.948} C_DIS
LIN {X -0.267,Y -501.841,Z 628.647,A 0.000,B 0.000,C 90.000,E1 332.487} C_DIS
LIN {X -0.139,Y -505.498,Z 628.634,A 0.000,B 0.000,C 90.000,E1 330.078} C_DIS
LIN {X 0.073,Y -510.270,Z 628.619,A 0.000,B 0.000,C 90.000,E1 327.375} C_DIS
LIN {X -0.143,Y -513.078,Z 628.612,A 0.000,B 0.000,C 90.000,E1 326.215} C_DIS
LIN {X 0.120,Y -514.753,Z 628.609,A 0.000,B 0.000,C 90.000,E1 325.595} C_DIS
LIN {X 0.045,Y -515.781,Z 628.607,A 0.000,B 0.000,C 90.000,E1 325.308} C_DIS
LIN {X 0.092,Y -517.140,Z 628.606,A 0.000,B 0.000,C 90.000,E1 325.022} C_DIS
LIN {X -0.102,Y -518.899,Z 628.603,A 0.000,B 0.000,C 90.000,E1 324.609} C_DIS
LIN {X 0.187,Y -521.200,Z 628.601,A 0.000,B 0.000,C 90.000,E1 324.196} C_DIS
LIN {X 0.060,Y -524.142,Z 628.599,A 0.000,B 0.000,C 90.000,E1 323.829} C_DIS
LIN {X 0.065,Y -528.756,Z 628.596,A 0.000,B 0.000,C 90.000,E1 323.336} C_DIS
LIN {X 0.159,Y -533.032,Z 628.594,A 0.000,B 0.000,C 90.000,E1 322.924} C_DIS
LIN {X 0.235,Y -544.583,Z 628.589,A 0.000,B 0.000,C 90.000,E1 321.984} C_DIS
LIN {X 0.226,Y -559.015,Z 628.582,A 0.000,B 0.000,C 90.000,E1 320.803} C_DIS
LIN {X -0.140,Y -573.114,Z 628.576,A 0.000,B 0.000,C 90.000,E1 319.666} C_DIS
LIN {X 0.212,Y -581.497,Z 628.572,A 0.000,B 0.000,C 90.000,E1 318.933} C_DIS
LIN {X -0.086,Y -588.267,Z 628.569,A 0.000,B 0.000,C 90.000,E1 318.366} C_DIS
LIN {X -0.043,Y -597.600,Z 628.564,A 0.000,B 0.000,C 90.000,E1 317.514} C_DIS
LIN {X 0.206,Y -601.260,Z 628.562,A 0.000,B 0.000,C 90.000,E1 317.148} C_DIS
LIN {X 0.180,Y -605.058,Z 628.560,A 0.000,B 0.000,C 90.000,E1 316.782} C_DIS
LIN {X -0.039,Y -609.951,Z 628.557,A 0.000,B 0.000,C 90.000,E1 316.296} C_DIS
LIN {X -0.364,Y -614.729,Z 628.554,A 0.000,B 0.000,C 90.000,E1 315.810} C_DIS
LIN {X 0.178,Y -619.299,Z 628.552,A 0.000,B 0.000,C 90.000,E1 315.243} C_DIS
LIN {X -0.123,Y -623.578,Z 628.549,A 0.000,B 0.000,C 90.000,E1 314.757} C_DIS
LIN {X 0.363,Y -629.686,Z 628.544,A 0.000,B 0.000,C 90.000,E1 313.947} C_DIS
LIN {X 0.016,Y -635.420,Z 628.540,A 0.000,B 0.000,C 90.000,E1 313.218} C_DIS
LIN {X 0.187,Y -641.052,Z 628.536,A 0.000,B 0.000,C 90.000,E1 312.447} C_DIS
LIN {X -0.073,Y -647.348,Z 628.531,A 0.000,B 0.000,C 90.000,E1 311.595} C_DIS
LIN {X -0.262,Y -654.140,Z 628.526,A 0.000,B 0.000,C 90.000,E1 310.620} C_DIS
LIN {X 0.140,Y -657.257,Z 628.523,A 0.000,B 0.000,C 90.000,E1 310.092} C_DIS
LIN {X -0.364,Y -660.159,Z 628.520,A 0.000,B 0.000,C 90.000,E1 309.644} C_DIS
LIN {X 0.113,Y -663.438,Z 628.517,A 0.000,B 0.000,C 90.000,E1 308.991} C_DIS
LIN {X -0.355,Y -665.888,Z 628.514,A 0.000,B 0.000,C 90.000,E1 308.543} C_DIS
LIN {X 0.206,Y -670.275,Z 628.509,A 0.000,B 0.000,C 90.000,E1 307.523} C_DIS
LIN {X -0.229,Y -672.299,Z 628.506,A 0.000,B 0.000,C 90.000,E1 307.076} C_DIS
LIN {X 0.416,Y -675.170,Z 628.502,A 0.000,B 0.000,C 90.000,E1 306.297} C_DIS
LIN {X 0.150,Y -677.751,Z 628.498,A 0.000,B 0.000,C 90.000,E1 305.598} C_DIS
LIN {X -0.094,Y -680.994,Z 628.493,A 0.000,B 0.000,C 90.000,E1 304.659} C_DIS
LIN {X -0.128,Y -684.050,Z 628.487,A 0.000,B 0.000,C 90.000,E1 303.706} C_DIS
LIN {X 0.087,Y -688.435,Z 628.479,A 0.000,B 0.000,C 90.000,E1 302.260} C_DIS
LIN {X 0.018,Y -691.864,Z 628.473,A 0.000,B 0.000,C 90.000,E1 301.082} C_DIS
LIN {X 0.125,Y -694.512,Z 628.467,A 0.000,B 0.000,C 90.000,E1 300.129} C_DIS
LIN {X 0.165,Y -697.528,Z 628.461,A 0.000,B 0.000,C 90.000,E1 298.949} C_DIS
LIN {X -0.015,Y -699.798,Z 628.456,A 0.000,B 0.000,C 90.000,E1 298.025} C_DIS
LIN {X -0.150,Y -701.286,Z 628.452,A 0.000,B 0.000,C 90.000,E1 297.334} C_DIS
LIN {X -0.223,Y -702.234,Z 628.449,A 0.000,B 0.000,C 90.000,E1 296.873} C_DIS
LIN {X 0.335,Y -703.001,Z 628.447,A 0.000,B 0.000,C 90.000,E1 296.360} C_DIS
LIN {X -0.043,Y -703.352,Z 628.444,A 0.000,B 0.000,C 90.000,E1 295.924} C_DIS
LIN {X 0.242,Y -703.473,Z 628.443,A 0.000,B 0.000,C 90.000,E1 295.668} C_DIS
LIN {X -0.110,Y -703.126,Z 628.441,A 0.000,B 0.000,C 90.000,E1 295.463} C_DIS
LIN {X 0.156,Y -702.050,Z 628.439,A 0.000,B 0.000,C 90.000,E1 294.975} C_DIS
LIN {X -0.341,Y -701.576,Z 628.438,A 0.000,B 0.000,C 90.000,E1 294.899} C_DIS
LIN {X -0.064,Y -699.916,Z 628.437,A 0.000,B 0.000,C 90.000,E1 294.643} C_DIS
LIN {X 0.053,Y -696.961,Z 628.435,A 0.000,B 0.000,C 90.000,E1 294.283} C_DIS
LIN {X 0.184,Y -695.628,Z 628.434,A 0.000,B 0.000,C 90.000,E1 294.155} C_DIS
LIN {X -0.320,Y -693.452,Z 628.434,A 0.000,B 0.000,C 90.000,E1 294.079} C_DIS
LIN {X -0.096,Y -685.571,Z 628.432,A 0.000,B 0.000,C 90.000,E1 293.770} C_DIS
LIN {X 0.098,Y -683.533,Z 628.432,A 0.000,B 0.000,C 90.000,E1 293.695} C_DIS
LIN {X 0.016,Y -680.558,Z 628.431,A 0.000,B 0.000,C 90.000,E1 293.643} C_DIS
LIN {X 0.354,Y -673.965,Z 628.431,A 0.000,B 0.000,C 90.000,E1 293.515} C_DIS
LIN {X 0.190,Y -667.102,Z 628.430,A 0.000,B 0.000,C 90.000,E1 293.462} C_DIS
LIN {X -0.134,Y -650.234,Z 628.429,A 0.000,B 0.000,C 90.000,E1 293.259} C_DIS
LIN {X -0.007,Y -640.452,Z 628.428,A 0.000,B 0.000,C 90.000,E1 293.078} C_DIS
LIN {X -0.338,Y -630.452,Z 628.427,A 0.000,B 0.000,C 90.000,E1 292.898} C_DIS
LIN {X -0.197,Y -620.956,Z 628.426,A 0.000,B 0.000,C 90.000,E1 292.642} C_DIS
LIN {X -0.024,Y -600.347,Z 628.422,A 0.000,B 0.000,C 90.000,E1 292.025} C_DIS
LIN {X 0.090,Y -579.469,Z 628.419,A 0.000,B 0.000,C 90.000,E1 291.354} C_DIS
LIN {X 0.054,Y -571.841,Z 628.418,A 0.000,B 0.000,C 90.000,E1 291.153} C_DIS
LIN {X -0.067,Y -564.113,Z 628.416,A 0.000,B 0.000,C 90.000,E1 290.918} C_DIS
LIN {X -0.308,Y -559.545,Z 628.415,A 0.000,B 0.000,C 90.000,E1 290.737} C_DIS
LIN {X 0.259,Y -557.141,Z 628.414,A 0.000,B 0.000,C 90.000,E1 290.482} C_DIS
LIN {X 0.223,Y -557.109,Z 628.414,A 0.000,B 0.000,C 90.000,E1 290.482} C_DIS
LIN {X 0.153,Y -556.482,Z 628.413,A 0.000,B 0.000,C 90.000,E1 290.301} C_DIS
LIN {X -0.266,Y -556.154,Z 628.411,A 0.000,B 0.000,C 90.000,E1 290.066} C_DIS
LIN {X 0.026,Y -555.983,Z 628.410,A 0.000,B 0.000,C 90.000,E1 289.758} C_DIS
LIN {X 0.283,Y -556.159,Z 628.405,A 0.000,B 0.000,C 90.000,E1 288.906} C_DIS
LIN {X 0.029,Y -556.177,Z 628.399,A 0.000,B 0.000,C 90.000,E1 287.819} C_DIS
LIN {X -0.231,Y -555.909,Z 628.393,A 0.000,B 0.000,C 90.000,E1 286.732} C_DIS
LIN {X -0.120,Y -555.592,Z 628.387,A 0.000,B 0.000,C 90.000,E1 285.607} C_DIS
LIN {X -0.008,Y -555.032,Z 628.380,A 0.000,B 0.000,C 90.000,E1 284.481} C_DIS
LIN {X 0.220,Y -554.336,Z 628.373,A 0.000,B 0.000,C 90.000,E1 283.063} C_DIS
LIN {X -0.104,Y -553.534,Z 628.363,A 0.000,B 0.000,C 90.000,E1 281.422} C_DIS
LIN {X 0.116,Y -552.631,Z 628.353,A 0.000,B 0.000,C 90.000,E1 279.443} C_DIS
LIN {X 0.230,Y -551.786,Z 628.342,A 0.000,B 0.000,C 90.000,E1 277.473} C_DIS
LIN {X 0.249,Y -550.985,Z 628.331,A 0.000,B 0.000,C 90.000,E1 275.511} C_DIS
LIN {X 0.189,Y -550.422,Z 628.320,A 0.000,B 0.000,C 90.000,E1 273.555} C_DIS
LIN {X 0.067,Y -549.900,Z 628.309,A 0.000,B 0.000,C 90.000,E1 271.604} C_DIS
LIN {X -0.210,Y -549.489,Z 628.301,A 0.000,B 0.000,C 90.000,E1 270.229} C_DIS
LIN {X 0.108,Y -548.742,Z 628.292,A 0.000,B 0.000,C 90.000,E1 268.511} C_DIS
LIN {X -0.103,Y -548.053,Z 628.282,A 0.000,B 0.000,C 90.000,E1 266.846} C_DIS
LIN {X 0.230,Y -547.140,Z 628.273,A 0.000,B 0.000,C 90.000,E1 265.122} C_DIS
LIN {X 0.043,Y -546.050,Z 628.264,A 0.000,B 0.000,C 90.000,E1 263.451} C_DIS
LIN {X 0.261,Y -545.101,Z 628.257,A 0.000,B 0.000,C 90.000,E1 262.299} C_DIS
LIN {X 0.082,Y -543.560,Z 628.250,A 0.000,B 0.000,C 90.000,E1 260.905} C_DIS
LIN {X 0.045,Y -541.515,Z 628.239,A 0.000,B 0.000,C 90.000,E1 258.926} C_DIS
LIN {X -0.015,Y -540.050,Z 628.229,A 0.000,B 0.000,C 90.000,E1 257.229} C_DIS
LIN {X 0.009,Y -538.667,Z 628.220,A 0.000,B 0.000,C 90.000,E1 255.519} C_DIS
LIN {X -0.122,Y -537.584,Z 628.213,A 0.000,B 0.000,C 90.000,E1 254.393} C_DIS
LIN {X -0.028,Y -535.734,Z 628.204,A 0.000,B 0.000,C 90.000,E1 252.670} C_DIS
LIN {X 0.143,Y -534.330,Z 628.196,A 0.000,B 0.000,C 90.000,E1 251.221} C_DIS
LIN {X 0.066,Y -533.407,Z 628.191,A 0.000,B 0.000,C 90.000,E1 250.369} C_DIS
LIN {X -0.124,Y -531.429,Z 628.183,A 0.000,B 0.000,C 90.000,E1 248.954} C_DIS
LIN {X -0.044,Y -529.720,Z 628.177,A 0.000,B 0.000,C 90.000,E1 247.794} C_DIS
LIN {X 0.205,Y -527.807,Z 628.170,A 0.000,B 0.000,C 90.000,E1 246.613} C_DIS
LIN {X 0.110,Y -525.123,Z 628.162,A 0.000,B 0.000,C 90.000,E1 245.177} C_DIS
LIN {X -0.128,Y -523.366,Z 628.157,A 0.000,B 0.000,C 90.000,E1 244.332} C_DIS
LIN {X -0.081,Y -520.211,Z 628.149,A 0.000,B 0.000,C 90.000,E1 242.871} C_DIS
LIN {X -0.199,Y -516.359,Z 628.140,A 0.000,B 0.000,C 90.000,E1 241.129} C_DIS
LIN {X 0.093,Y -513.712,Z 628.133,A 0.000,B 0.000,C 90.000,E1 239.921} C_DIS
LIN {X -0.005,Y -510.179,Z 628.125,A 0.000,B 0.000,C 90.000,E1 238.456} C_DIS
LIN {X 0.097,Y -506.550,Z 628.117,A 0.000,B 0.000,C 90.000,E1 236.962} C_DIS
LIN {X 0.124,Y -502.783,Z 628.108,A 0.000,B 0.000,C 90.000,E1 235.468} C_DIS
LIN {X 0.069,Y -499.715,Z 628.102,A 0.000,B 0.000,C 90.000,E1 234.276} C_DIS
LIN {X 0.265,Y -492.603,Z 628.087,A 0.000,B 0.000,C 90.000,E1 231.537} C_DIS
LIN {X -0.032,Y -489.547,Z 628.080,A 0.000,B 0.000,C 90.000,E1 230.356} C_DIS
LIN {X -0.085,Y -485.079,Z 628.070,A 0.000,B 0.000,C 90.000,E1 228.528} C_DIS
LIN {X 0.088,Y -480.544,Z 628.059,A 0.000,B 0.000,C 90.000,E1 226.662} C_DIS
LIN {X -0.084,Y -475.206,Z 628.047,A 0.000,B 0.000,C 90.000,E1 224.514} C_DIS
LIN {X -0.049,Y -470.191,Z 628.035,A 0.000,B 0.000,C 90.000,E1 222.324} C_DIS
LIN {X 0.022,Y -466.788,Z 628.026,A 0.000,B 0.000,C 90.000,E1 220.744} C_DIS
LIN {X 0.011,Y -464.096,Z 628.019,A 0.000,B 0.000,C 90.000,E1 219.483} C_DIS
LIN {X -0.183,Y -460.044,Z 628.009,A 0.000,B 0.000,C 90.000,E1 217.604} C_DIS
LIN {X -0.099,Y -455.600,Z 627.996,A 0.000,B 0.000,C 90.000,E1 215.358} C_DIS
LIN {X 0.071,Y -451.485,Z 627.984,A 0.000,B 0.000,C 90.000,E1 213.086} C_DIS
LIN {X -0.115,Y -447.314,Z 627.971,A 0.000,B 0.000,C 90.000,E1 210.846} C_DIS
LIN {X 0.061,Y -443.908,Z 627.961,A 0.000,B 0.000,C 90.000,E1 208.871} C_DIS
LIN {X -0.097,Y -440.996,Z 627.951,A 0.000,B 0.000,C 90.000,E1 207.257} C_DIS
LIN {X 0.053,Y -438.747,Z 627.944,A 0.000,B 0.000,C 90.000,E1 205.924} C_DIS
LIN {X -0.156,Y -434.553,Z 627.931,A 0.000,B 0.000,C 90.000,E1 203.643} C_DIS
LIN {X -0.064,Y -431.657,Z 627.922,A 0.000,B 0.000,C 90.000,E1 201.972} C_DIS
LIN {X 0.178,Y -428.253,Z 627.911,A 0.000,B 0.000,C 90.000,E1 199.939} C_DIS
LIN {X 0.046,Y -424.961,Z 627.900,A 0.000,B 0.000,C 90.000,E1 197.946} C_DIS
LIN {X 0.057,Y -422.366,Z 627.890,A 0.000,B 0.000,C 90.000,E1 196.260} C_DIS
LIN {X -0.049,Y -419.313,Z 627.879,A 0.000,B 0.000,C 90.000,E1 194.245} C_DIS
LIN {X 0.028,Y -416.651,Z 627.870,A 0.000,B 0.000,C 90.000,E1 192.535} C_DIS
LIN {X 0.134,Y -412.171,Z 627.853,A 0.000,B 0.000,C 90.000,E1 189.443} C_DIS
LIN {X -0.129,Y -410.294,Z 627.845,A 0.000,B 0.000,C 90.000,E1 188.106} C_DIS
LIN {X -0.059,Y -407.858,Z 627.835,A 0.000,B 0.000,C 90.000,E1 186.372} C_DIS
LIN {X -0.148,Y -404.320,Z 627.820,A 0.000,B 0.000,C 90.000,E1 183.612} C_DIS
LIN {X 0.048,Y -401.654,Z 627.806,A 0.000,B 0.000,C 90.000,E1 181.146} C_DIS
LIN {X 0.010,Y -398.675,Z 627.787,A 0.000,B 0.000,C 90.000,E1 177.650} C_DIS
LIN {X -0.081,Y -396.841,Z 627.767,A 0.000,B 0.000,C 90.000,E1 174.147} C_DIS
LIN {X -0.023,Y -396.110,Z 627.752,A 0.000,B 0.000,C 90.000,E1 171.319} C_DIS
LIN {X -0.162,Y -395.784,Z 627.738,A 0.000,B 0.000,C 90.000,E1 168.870} C_DIS
LIN {X 0.219,Y -395.902,Z 627.722,A 0.000,B 0.000,C 90.000,E1 165.992} C_DIS
LIN {X -0.054,Y -396.129,Z 627.713,A 0.000,B 0.000,C 90.000,E1 164.267} C_DIS
LIN {X -0.191,Y -396.595,Z 627.699,A 0.000,B 0.000,C 90.000,E1 161.819} C_DIS
LIN {X 0.128,Y -397.271,Z 627.683,A 0.000,B 0.000,C 90.000,E1 158.954} C_DIS
LIN {X 0.166,Y -397.987,Z 627.670,A 0.000,B 0.000,C 90.000,E1 156.485} C_DIS
LIN {X -0.058,Y -398.616,Z 627.658,A 0.000,B 0.000,C 90.000,E1 154.409} C_DIS
LIN {X 0.083,Y -399.287,Z 627.646,A 0.000,B 0.000,C 90.000,E1 152.281} C_DIS
LIN {X 0.002,Y -399.829,Z 627.636,A 0.000,B 0.000,C 90.000,E1 150.539} C_DIS
LIN {X -0.135,Y -400.434,Z 627.625,A 0.000,B 0.000,C 90.000,E1 148.456} C_DIS
LIN {X -0.037,Y -401.072,Z 627.613,A 0.000,B 0.000,C 90.000,E1 146.342} C_DIS
LIN {X -0.145,Y -401.971,Z 627.599,A 0.000,B 0.000,C 90.000,E1 143.909} C_DIS
LIN {X -0.016,Y -402.689,Z 627.590,A 0.000,B 0.000,C 90.000,E1 142.145} C_DIS
LIN {X -0.264,Y -403.349,Z 627.580,A 0.000,B 0.000,C 90.000,E1 140.436} C_DIS
LIN {X 0.021,Y -404.143,Z 627.566,A 0.000,B 0.000,C 90.000,E1 137.957} C_DIS
LIN {X 0.036,Y -404.608,Z 627.557,A 0.000,B 0.000,C 90.000,E1 136.215} C_DIS
LIN {X 0.183,Y -405.245,Z 627.545,A 0.000,B 0.000,C 90.000,E1 134.109} C_DIS
LIN {X 0.026,Y -406.290,Z 627.530,A 0.000,B 0.000,C 90.000,E1 131.353} C_DIS
LIN {X -0.004,Y -407.483,Z 627.518,A 0.000,B 0.000,C 90.000,E1 129.277} C_DIS
LIN {X -0.028,Y -408.161,Z 627.514,A 0.000,B 0.000,C 90.000,E1 128.588} C_DIS
LIN {X 0.206,Y -408.434,Z 627.513,A 0.000,B 0.000,C 90.000,E1 128.382} C_DIS
LIN {X -0.074,Y -414.174,Z 627.502,A 0.000,B 0.000,C 90.000,E1 126.423} C_DIS
LIN {X -0.113,Y -414.193,Z 627.502,A 0.000,B 0.000,C 90.000,E1 126.423} C_DIS
LIN {X -0.015,Y -416.923,Z 627.501,A 0.000,B 0.000,C 90.000,E1 126.091} C_DIS
LIN {X -0.089,Y -421.516,Z 627.498,A 0.000,B 0.000,C 90.000,E1 125.724} C_DIS
LIN {X -0.061,Y -428.108,Z 627.496,A 0.000,B 0.000,C 90.000,E1 125.311} C_DIS
LIN {X 0.273,Y -448.192,Z 627.490,A 0.000,B 0.000,C 90.000,E1 124.119} C_DIS
LIN {X 0.094,Y -456.435,Z 627.487,A 0.000,B 0.000,C 90.000,E1 123.658} C_DIS
LIN {X -0.002,Y -464.606,Z 627.484,A 0.000,B 0.000,C 90.000,E1 123.166} C_DIS
LIN {X -0.074,Y -474.314,Z 627.481,A 0.000,B 0.000,C 90.000,E1 122.546} C_DIS
LIN {X -0.019,Y -482.270,Z 627.478,A 0.000,B 0.000,C 90.000,E1 122.005} C_DIS
LIN {X -0.015,Y -491.555,Z 627.474,A 0.000,B 0.000,C 90.000,E1 121.337} C_DIS
LIN {X -0.251,Y -500.780,Z 627.470,A 0.000,B 0.000,C 90.000,E1 120.669} C_DIS
LIN {X 0.269,Y -505.260,Z 627.468,A 0.000,B 0.000,C 90.000,E1 120.256} C_DIS
LIN {X 0.114,Y -512.585,Z 627.465,A 0.000,B 0.000,C 90.000,E1 119.667} C_DIS
LIN {X -0.074,Y -518.305,Z 627.462,A 0.000,B 0.000,C 90.000,E1 119.205} C_DIS
LIN {X -0.220,Y -525.158,Z 627.459,A 0.000,B 0.000,C 90.000,E1 118.615} C_DIS
LIN {X -0.212,Y -530.681,Z 627.456,A 0.000,B 0.000,C 90.000,E1 118.103} C_DIS
LIN {X -0.283,Y -534.718,Z 627.454,A 0.000,B 0.000,C 90.000,E1 117.719} C_DIS
LIN {X -0.066,Y -539.548,Z 627.451,A 0.000,B 0.000,C 90.000,E1 117.206} C_DIS
LIN {X -0.091,Y -544.177,Z 627.448,A 0.000,B 0.000,C 90.000,E1 116.693} C_DIS
LIN {X 0.060,Y -548.516,Z 627.445,A 0.000,B 0.000,C 90.000,E1 116.155} C_DIS
LIN {X -0.052,Y -553.223,Z 627.442,A 0.000,B 0.000,C 90.000,E1 115.515} C_DIS
LIN {X -0.116,Y -557.644,Z 627.438,A 0.000,B 0.000,C 90.000,E1 114.823} C_DIS
LIN {X -0.137,Y -561.549,Z 627.434,A 0.000,B 0.000,C 90.000,E1 114.131} C_DIS
LIN {X 0.295,Y -565.720,Z 627.429,A 0.000,B 0.000,C 90.000,E1 113.259} C_DIS
LIN {X -0.058,Y -569.940,Z 627.424,A 0.000,B 0.000,C 90.000,E1 112.333} C_DIS
LIN {X -0.281,Y -573.351,Z 627.420,A 0.000,B 0.000,C 90.000,E1 111.535} C_DIS
LIN {X 0.276,Y -576.455,Z 627.415,A 0.000,B 0.000,C 90.000,E1 110.663} C_DIS
LIN {X 0.283,Y -578.428,Z 627.412,A 0.000,B 0.000,C 90.000,E1 110.120} C_DIS
LIN {X 0.146,Y -581.128,Z 627.407,A 0.000,B 0.000,C 90.000,E1 109.322} C_DIS
LIN {X -0.155,Y -583.536,Z 627.403,A 0.000,B 0.000,C 90.000,E1 108.544} C_DIS
LIN {X -0.025,Y -586.387,Z 627.397,A 0.000,B 0.000,C 90.000,E1 107.457} C_DIS
LIN {X 0.055,Y -587.718,Z 627.394,A 0.000,B 0.000,C 90.000,E1 106.913} C_DIS
LIN {X 0.016,Y -591.630,Z 627.385,A 0.000,B 0.000,C 90.000,E1 105.315} C_DIS
LIN {X 0.199,Y -597.064,Z 627.373,A 0.000,B 0.000,C 90.000,E1 103.175} C_DIS
LIN {X -0.086,Y -600.494,Z 627.366,A 0.000,B 0.000,C 90.000,E1 101.883} C_DIS
LIN {X -0.158,Y -603.271,Z 627.360,A 0.000,B 0.000,C 90.000,E1 100.838} C_DIS
LIN {X 0.144,Y -606.632,Z 627.353,A 0.000,B 0.000,C 90.000,E1 99.500} C_DIS
LIN {X -0.103,Y -609.721,Z 627.346,A 0.000,B 0.000,C 90.000,E1 98.219} C_DIS
LIN {X -0.128,Y -613.218,Z 627.337,A 0.000,B 0.000,C 90.000,E1 96.663} C_DIS
LIN {X 0.246,Y -615.771,Z 627.330,A 0.000,B 0.000,C 90.000,E1 95.334} C_DIS
LIN {X 0.285,Y -618.353,Z 627.321,A 0.000,B 0.000,C 90.000,E1 93.784} C_DIS
LIN {X -0.292,Y -619.974,Z 627.315,A 0.000,B 0.000,C 90.000,E1 92.808} C_DIS
LIN {X -0.232,Y -621.316,Z 627.310,A 0.000,B 0.000,C 90.000,E1 91.776} C_DIS
LIN {X -0.173,Y -622.416,Z 627.304,A 0.000,B 0.000,C 90.000,E1 90.745} C_DIS
LIN {X 0.198,Y -623.078,Z 627.300,A 0.000,B 0.000,C 90.000,E1 89.943} C_DIS
LIN {X -0.049,Y -623.548,Z 627.296,A 0.000,B 0.000,C 90.000,E1 89.198} C_DIS
LIN {X -0.293,Y -623.894,Z 627.291,A 0.000,B 0.000,C 90.000,E1 88.453} C_DIS
LIN {X 0.108,Y -623.998,Z 627.287,A 0.000,B 0.000,C 90.000,E1 87.650} C_DIS
LIN {X 0.228,Y -623.944,Z 627.281,A 0.000,B 0.000,C 90.000,E1 86.617} C_DIS
LIN {X 0.016,Y -623.753,Z 627.277,A 0.000,B 0.000,C 90.000,E1 85.869} C_DIS
LIN {X -0.171,Y -623.099,Z 627.270,A 0.000,B 0.000,C 90.000,E1 84.609} C_DIS
LIN {X -0.020,Y -622.398,Z 627.264,A 0.000,B 0.000,C 90.000,E1 83.571} C_DIS
LIN {X 0.121,Y -621.519,Z 627.259,A 0.000,B 0.000,C 90.000,E1 82.534} C_DIS
LIN {X -0.049,Y -620.665,Z 627.254,A 0.000,B 0.000,C 90.000,E1 81.781} C_DIS
LIN {X 0.155,Y -619.235,Z 627.249,A 0.000,B 0.000,C 90.000,E1 80.735} C_DIS
LIN {X 0.106,Y -617.202,Z 627.242,A 0.000,B 0.000,C 90.000,E1 79.454} C_DIS
LIN {X 0.021,Y -614.905,Z 627.234,A 0.000,B 0.000,C 90.000,E1 78.173} C_DIS
LIN {X 0.018,Y -612.359,Z 627.227,A 0.000,B 0.000,C 90.000,E1 76.881} C_DIS
LIN {X 0.220,Y -610.107,Z 627.221,A 0.000,B 0.000,C 90.000,E1 75.825} C_DIS
LIN {X -0.049,Y -607.799,Z 627.216,A 0.000,B 0.000,C 90.000,E1 74.810} C_DIS
LIN {X -0.025,Y -604.690,Z 627.208,A 0.000,B 0.000,C 90.000,E1 73.504} C_DIS
LIN {X -0.085,Y -602.687,Z 627.204,A 0.000,B 0.000,C 90.000,E1 72.725} C_DIS
LIN {X 0.307,Y -599.744,Z 627.198,A 0.000,B 0.000,C 90.000,E1 71.638} C_DIS
LIN {X -0.079,Y -598.088,Z 627.195,A 0.000,B 0.000,C 90.000,E1 71.148} C_DIS
LIN {X 0.093,Y -596.392,Z 627.192,A 0.000,B 0.000,C 90.000,E1 70.604} C_DIS
LIN {X -0.060,Y -593.594,Z 627.188,A 0.000,B 0.000,C 90.000,E1 69.826} C_DIS
LIN {X -0.040,Y -590.521,Z 627.184,A 0.000,B 0.000,C 90.000,E1 69.028} C_DIS
LIN {X -0.052,Y -587.235,Z 627.179,A 0.000,B 0.000,C 90.000,E1 68.230} C_DIS
LIN {X -0.228,Y -582.574,Z 627.173,A 0.000,B 0.000,C 90.000,E1 67.177} C_DIS
LIN {X -0.172,Y -578.045,Z 627.168,A 0.000,B 0.000,C 90.000,E1 66.230} C_DIS
LIN {X -0.012,Y -574.611,Z 627.164,A 0.000,B 0.000,C 90.000,E1 65.537} C_DIS
LIN {X 0.196,Y -571.724,Z 627.161,A 0.000,B 0.000,C 90.000,E1 64.973} C_DIS
LIN {X -0.183,Y -567.694,Z 627.157,A 0.000,B 0.000,C 90.000,E1 64.332} C_DIS
LIN {X -0.084,Y -563.289,Z 627.154,A 0.000,B 0.000,C 90.000,E1 63.640} C_DIS
LIN {X 0.033,Y -559.351,Z 627.151,A 0.000,B 0.000,C 90.000,E1 63.076} C_DIS
LIN {X 0.264,Y -553.880,Z 627.147,A 0.000,B 0.000,C 90.000,E1 62.359} C_DIS
LIN {X -0.067,Y -550.381,Z 627.144,A 0.000,B 0.000,C 90.000,E1 61.975} C_DIS
LIN {X -0.113,Y -545.217,Z 627.141,A 0.000,B 0.000,C 90.000,E1 61.435} C_DIS
LIN {X 0.143,Y -542.090,Z 627.140,A 0.000,B 0.000,C 90.000,E1 61.129} C_DIS
LIN {X 0.190,Y -540.017,Z 627.139,A 0.000,B 0.000,C 90.000,E1 60.923} C_DIS
LIN {X 0.084,Y -534.161,Z 627.136,A 0.000,B 0.000,C 90.000,E1 60.461} C_DIS
LIN {X 0.233,Y -530.709,Z 627.135,A 0.000,B 0.000,C 90.000,E1 60.205} C_DIS
LIN {X -0.082,Y -529.209,Z 627.134,A 0.000,B 0.000,C 90.000,E1 60.127} C_DIS
LIN {X -0.077,Y -522.531,Z 627.132,A 0.000,B 0.000,C 90.000,E1 59.715} C_DIS
LIN {X 0.193,Y -517.827,Z 627.130,A 0.000,B 0.000,C 90.000,E1 59.410} C_DIS
LIN {X 0.008,Y -511.372,Z 627.128,A 0.000,B 0.000,C 90.000,E1 59.076} C_DIS
LIN {X -0.216,Y -502.587,Z 627.126,A 0.000,B 0.000,C 90.000,E1 58.663} C_DIS
LIN {X 0.060,Y -484.049,Z 627.121,A 0.000,B 0.000,C 90.000,E1 57.709} C_DIS
LIN {X -0.190,Y -462.014,Z 627.115,A 0.000,B 0.000,C 90.000,E1 56.628} C_DIS
LIN {X -0.055,Y -441.485,Z 627.108,A 0.000,B 0.000,C 90.000,E1 55.515} C_DIS
LIN {X -0.099,Y -441.426,Z 627.108,A 0.000,B 0.000,C 90.000,E1 55.515} C_DIS
LIN {X 0.245,Y -432.731,Z 627.086,A 0.000,B 0.000,C 90.000,E1 51.457} C_DIS
LIN {X 0.160,Y -431.528,Z 627.082,A 0.000,B 0.000,C 90.000,E1 50.803} C_DIS
LIN {X 0.027,Y -426.216,Z 627.070,A 0.000,B 0.000,C 90.000,E1 48.609} C_DIS
LIN {X 0.060,Y -426.741,Z 627.064,A 0.000,B 0.000,C 90.000,E1 47.472} C_DIS
LIN {X 0.026,Y -427.237,Z 627.056,A 0.000,B 0.000,C 90.000,E1 46.134} C_DIS
LIN {X 0.052,Y -427.900,Z 627.043,A 0.000,B 0.000,C 90.000,E1 43.785} C_DIS
LIN {X 0.106,Y -428.775,Z 627.030,A 0.000,B 0.000,C 90.000,E1 41.434} C_DIS
LIN {X 0.024,Y -429.662,Z 627.019,A 0.000,B 0.000,C 90.000,E1 39.439} C_DIS
LIN {X -0.280,Y -430.485,Z 627.010,A 0.000,B 0.000,C 90.000,E1 37.810} C_DIS
LIN {X 0.109,Y -431.226,Z 627.001,A 0.000,B 0.000,C 90.000,E1 36.091} C_DIS
LIN {X -0.095,Y -432.022,Z 626.990,A 0.000,B 0.000,C 90.000,E1 34.119} C_DIS
LIN {X 0.185,Y -432.627,Z 626.980,A 0.000,B 0.000,C 90.000,E1 32.418} C_DIS
LIN {X -0.104,Y -433.285,Z 626.969,A 0.000,B 0.000,C 90.000,E1 30.463} C_DIS
LIN {X 0.169,Y -434.162,Z 626.956,A 0.000,B 0.000,C 90.000,E1 28.103} C_DIS
LIN {X 0.064,Y -435.127,Z 626.943,A 0.000,B 0.000,C 90.000,E1 25.796} C_DIS
LIN {X -0.207,Y -436.058,Z 626.931,A 0.000,B 0.000,C 90.000,E1 23.515} C_DIS
LIN {X -0.072,Y -436.842,Z 626.921,A 0.000,B 0.000,C 90.000,E1 21.844} C_DIS
LIN {X 0.075,Y -437.752,Z 626.912,A 0.000,B 0.000,C 90.000,E1 20.174} C_DIS
LIN {X 0.189,Y -438.737,Z 626.901,A 0.000,B 0.000,C 90.000,E1 18.181} C_DIS
LIN {X 0.031,Y -439.992,Z 626.888,A 0.000,B 0.000,C 90.000,E1 15.898} C_DIS
LIN {X -0.060,Y -441.208,Z 626.877,A 0.000,B 0.000,C 90.000,E1 13.939} C_DIS
LIN {X 0.082,Y -443.065,Z 626.863,A 0.000,B 0.000,C 90.000,E1 11.299} C_DIS
LIN {X -0.221,Y -445.515,Z 626.847,A 0.000,B 0.000,C 90.000,E1 8.398} C_DIS
LIN {X -0.103,Y -447.409,Z 626.836,A 0.000,B 0.000,C 90.000,E1 6.429} C_DIS
LIN {X 0.102,Y -449.753,Z 626.823,A 0.000,B 0.000,C 90.000,E1 4.131} C_DIS
LIN {X -0.094,Y -452.372,Z 626.810,A 0.000,B 0.000,C 90.000,E1 1.892} C_DIS
LIN {X -0.199,Y -456.421,Z 626.794,A 0.000,B 0.000,C 90.000,E1 358.854} C_DIS
LIN {X -0.219,Y -459.852,Z 626.781,A 0.000,B 0.000,C 90.000,E1 356.617} C_DIS
LIN {X 0.107,Y -462.978,Z 626.771,A 0.000,B 0.000,C 90.000,E1 354.666} C_DIS
LIN {X -0.069,Y -466.766,Z 626.758,A 0.000,B 0.000,C 90.000,E1 352.470} C_DIS
LIN {X 0.116,Y -470.000,Z 626.748,A 0.000,B 0.000,C 90.000,E1 350.557} C_DIS
LIN {X -0.102,Y -473.127,Z 626.737,A 0.000,B 0.000,C 90.000,E1 348.701} C_DIS
LIN {X 0.087,Y -475.853,Z 626.729,A 0.000,B 0.000,C 90.000,E1 347.117} C_DIS
LIN {X 0.136,Y -479.689,Z 626.716,A 0.000,B 0.000,C 90.000,E1 344.936} C_DIS
LIN {X 0.081,Y -483.784,Z 626.704,A 0.000,B 0.000,C 90.000,E1 342.779} C_DIS
LIN {X -0.184,Y -487.378,Z 626.694,A 0.000,B 0.000,C 90.000,E1 340.967} C_DIS
LIN {X 0.222,Y -490.342,Z 626.686,A 0.000,B 0.000,C 90.000,E1 339.390} C_DIS
LIN {X -0.060,Y -493.224,Z 626.677,A 0.000,B 0.000,C 90.000,E1 337.901} C_DIS
LIN {X 0.121,Y -495.315,Z 626.670,A 0.000,B 0.000,C 90.000,E1 336.666} C_DIS
LIN {X -0.129,Y -497.310,Z 626.664,A 0.000,B 0.000,C 90.000,E1 335.485} C_DIS
LIN {X -0.092,Y -499.623,Z 626.655,A 0.000,B 0.000,C 90.000,E1 333.973} C_DIS
LIN {X -0.240,Y -501.867,Z 626.647,A 0.000,B 0.000,C 90.000,E1 332.487} C_DIS
LIN {X -0.041,Y -504.561,Z 626.637,A 0.000,B 0.000,C 90.000,E1 330.667} C_DIS
LIN {X -0.273,Y -510.767,Z 626.617,A 0.000,B 0.000,C 90.000,E1 327.120} C_DIS
LIN {X 0.223,Y -513.532,Z 626.611,A 0.000,B 0.000,C 90.000,E1 325.881} C_DIS
LIN {X 0.065,Y -515.185,Z 626.607,A 0.000,B 0.000,C 90.000,E1 325.308} C_DIS
LIN {X -0.008,Y -516.375,Z 626.606,A 0.000,B 0.000,C 90.000,E1 325.022} C_DIS
LIN {X 0.164,Y -517.914,Z 626.603,A 0.000,B 0.000,C 90.000,E1 324.562} C_DIS
LIN {X 0.222,Y -520.134,Z 626.601,A 0.000,B 0.000,C 90.000,E1 324.116} C_DIS
LIN {X -0.011,Y -522.974,Z 626.598,A 0.000,B 0.000,C 90.000,E1 323.703} C_DIS
LIN {X -0.057,Y -525.173,Z 626.597,A 0.000,B 0.000,C 90.000,E1 323.417} C_DIS
LIN {X -0.056,Y -527.793,Z 626.595,A 0.000,B 0.000,C 90.000,E1 323.130} C_DIS
LIN {X 0.019,Y -532.982,Z 626.592,A 0.000,B 0.000,C 90.000,E1 322.637} C_DIS
LIN {X 0.022,Y -539.002,Z 626.590,A 0.000,B 0.000,C 90.000,E1 322.145} C_DIS
LIN {X 0.226,Y -546.248,Z 626.586,A 0.000,B 0.000,C 90.000,E1 321.537} C_DIS
LIN {X 0.180,Y -557.785,Z 626.581,A 0.000,B 0.000,C 90.000,E1 320.598} C_DIS
LIN {X -0.122,Y -574.966,Z 626.573,A 0.000,B 0.000,C 90.000,E1 319.218} C_DIS
LIN {X -0.150,Y -584.667,Z 626.569,A 0.000,B 0.000,C 90.000,E1 318.405} C_DIS
LIN {X -0.025,Y -596.832,Z 626.563,A 0.000,B 0.000,C 90.000,E1 317.310} C_DIS
LIN {X -0.033,Y -603.360,Z 626.560,A 0.000,B 0.000,C 90.000,E1 316.701} C_DIS
LIN {X 0.167,Y -609.479,Z 626.556,A 0.000,B 0.000,C 90.000,E1 316.053} C_DIS
LIN {X 0.226,Y -615.505,Z 626.552,A 0.000,B 0.000,C 90.000,E1 315.405} C_DIS
LIN {X -0.044,Y -619.981,Z 626.550,A 0.000,B 0.000,C 90.000,E1 314.919} C_DIS
LIN {X 0.318,Y -627.041,Z 626.545,A 0.000,B 0.000,C 90.000,E1 314.028} C_DIS
LIN {X 0.018,Y -631.969,Z 626.541,A 0.000,B 0.000,C 90.000,E1 313.419} C_DIS
LIN {X 0.092,Y -638.662,Z 626.536,A 0.000,B 0.000,C 90.000,E1 312.528} C_DIS
LIN {X -0.195,Y -645.151,Z 626.531,A 0.000,B 0.000,C 90.000,E1 311.676} C_DIS
LIN {X -0.368,Y -652.143,Z 626.526,A 0.000,B 0.000,C 90.000,E1 310.701} C_DIS
LIN {X -0.421,Y -656.093,Z 626.523,A 0.000,B 0.000,C 90.000,E1 310.092} C_DIS
LIN {X -0.008,Y -659.064,Z 626.520,A 0.000,B 0.000,C 90.000,E1 309.564} C_DIS
LIN {X -0.054,Y -662.430,Z 626.516,A 0.000,B 0.000,C 90.000,E1 308.955} C_DIS
LIN {X 0.029,Y -665.486,Z 626.513,A 0.000,B 0.000,C 90.000,E1 308.338} C_DIS
LIN {X 0.057,Y -670.028,Z 626.508,A 0.000,B 0.000,C 90.000,E1 307.363} C_DIS
LIN {X -0.264,Y -673.055,Z 626.504,A 0.000,B 0.000,C 90.000,E1 306.664} C_DIS
LIN {X -0.154,Y -675.783,Z 626.500,A 0.000,B 0.000,C 90.000,E1 305.931} C_DIS
LIN {X -0.266,Y -679.957,Z 626.493,A 0.000,B 0.000,C 90.000,E1 304.739} C_DIS
LIN {X 0.252,Y -683.843,Z 626.486,A 0.000,B 0.000,C 90.000,E1 303.499} C_DIS
LIN {X 0.099,Y -688.308,Z 626.478,A 0.000,B 0.000,C 90.000,E1 302.084} C_DIS
LIN {X -0.198,Y -691.733,Z 626.472,A 0.000,B 0.000,C 90.000,E1 300.924} C_DIS
LIN {X 0.152,Y -694.405,Z 626.466,A 0.000,B 0.000,C 90.000,E1 299.951} C_DIS
LIN {X -0.057,Y -696.911,Z 626.461,A 0.000,B 0.000,C 90.000,E1 299.027} C_DIS
LIN {X -0.242,Y -699.265,Z 626.456,A 0.000,B 0.000,C 90.000,E1 298.103} C_DIS
LIN {X -0.056,Y -700.846,Z 626.452,A 0.000,B 0.000,C 90.000,E1 297.385} C_DIS
LIN {X -0.134,Y -701.813,Z 626.450,A 0.000,B 0.000,C 90.000,E1 296.924} C_DIS
LIN {X 0.105,Y -702.611,Z 626.447,A 0.000,B 0.000,C 90.000,E1 296.437} C_DIS
LIN {X -0.245,Y -702.892,Z 626.446,A 0.000,B 0.000,C 90.000,E1 296.232} C_DIS
LIN {X 0.317,Y -703.165,Z 626.443,A 0.000,B 0.000,C 90.000,E1 295.720} C_DIS
LIN {X -0.339,Y -702.960,Z 626.442,A 0.000,B 0.000,C 90.000,E1 295.540} C_DIS
LIN {X 0.224,Y -701.895,Z 626.439,A 0.000,B 0.000,C 90.000,E1 295.027} C_DIS
LIN {X -0.133,Y -700.891,Z 626.438,A 0.000,B 0.000,C 90.000,E1 294.823} C_DIS
LIN {X 0.119,Y -697.005,Z 626.435,A 0.000,B 0.000,C 90.000,E1 294.335} C_DIS
LIN {X 0.250,Y -695.866,Z 626.435,A 0.000,B 0.000,C 90.000,E1 294.207} C_DIS
LIN {X 0.378,Y -694.106,Z 626.434,A 0.000,B 0.000,C 90.000,E1 294.079} C_DIS
LIN {X -0.145,Y -691.821,Z 626.433,A 0.000,B 0.000,C 90.000,E1 294.027} C_DIS
LIN {X 0.301,Y -685.941,Z 626.432,A 0.000,B 0.000,C 90.000,E1 293.770} C_DIS
LIN {X -0.056,Y -682.529,Z 626.432,A 0.000,B 0.000,C 90.000,E1 293.695} C_DIS
LIN {X -0.124,Y -673.886,Z 626.431,A 0.000,B 0.000,C 90.000,E1 293.567} C_DIS
LIN {X -0.279,Y -667.151,Z 626.431,A 0.000,B 0.000,C 90.000,E1 293.515} C_DIS
LIN {X 0.003,Y -650.321,Z 626.429,A 0.000,B 0.000,C 90.000,E1 293.259} C_DIS
LIN {X 0.136,Y -640.474,Z 626.428,A 0.000,B 0.000,C 90.000,E1 293.078} C_DIS
LIN {X -0.196,Y -630.480,Z 626.427,A 0.000,B 0.000,C 90.000,E1 292.898} C_DIS
LIN {X -0.073,Y -620.903,Z 626.426,A 0.000,B 0.000,C 90.000,E1 292.642} C_DIS
LIN {X 0.115,Y -600.395,Z 626.422,A 0.000,B 0.000,C 90.000,E1 292.025} C_DIS
LIN {X 0.214,Y -579.520,Z 626.419,A 0.000,B 0.000,C 90.000,E1 291.354} C_DIS
LIN {X 0.177,Y -571.810,Z 626.418,A 0.000,B 0.000,C 90.000,E1 291.153} C_DIS
LIN {X 0.076,Y -564.233,Z 626.416,A 0.000,B 0.000,C 90.000,E1 290.918} C_DIS
LIN {X -0.188,Y -559.629,Z 626.415,A 0.000,B 0.000,C 90.000,E1 290.737} C_DIS
LIN {X 0.235,Y -557.233,Z 626.414,A 0.000,B 0.000,C 90.000,E1 290.482} C_DIS
LIN {X 0.197,Y -557.199,Z 626.414,A 0.000,B 0.000,C 90.000,E1 290.482} C_DIS
LIN {X 0.115,Y -556.568,Z 626.413,A 0.000,B 0.000,C 90.000,E1 290.301} C_DIS
LIN {X -0.303,Y -556.241,Z 626.411,A 0.000,B 0.000,C 90.000,E1 290.066} C_DIS
LIN {X -0.010,Y -556.124,Z 626.410,A 0.000,B 0.000,C 90.000,E1 289.758} C_DIS
LIN {X 0.247,Y -556.277,Z 626.405,A 0.000,B 0.000,C 90.000,E1 288.906} C_DIS
LIN {X -0.006,Y -556.296,Z 626.399,A 0.000,B 0.000,C 90.000,E1 287.819} C_DIS
LIN {X 0.269,Y -556.029,Z 626.393,A 0.000,B 0.000,C 90.000,E1 286.677} C_DIS
LIN {X -0.151,Y -555.712,Z 626.387,A 0.000,B 0.000,C 90.000,E1 285.607} C_DIS
LIN {X -0.037,Y -555.153,Z 626.380,A 0.000,B 0.000,C 90.000,E1 284.481} C_DIS
LIN {X 0.193,Y -554.458,Z 626.373,A 0.000,B 0.000,C 90.000,E1 283.063} C_DIS
LIN {X -0.129,Y -553.656,Z 626.363,A 0.000,B 0.000,C 90.000,E1 281.422} C_DIS
LIN {X 0.066,Y -552.842,Z 626.354,A 0.000,B 0.000,C 90.000,E1 279.726} C_DIS
LIN {X 0.056,Y -552.113,Z 626.345,A 0.000,B 0.000,C 90.000,E1 278.049} C_DIS
LIN {X 0.035,Y -551.389,Z 626.335,A 0.000,B 0.000,C 90.000,E1 276.372} C_DIS
LIN {X -0.022,Y -550.693,Z 626.325,A 0.000,B 0.000,C 90.000,E1 274.416} C_DIS
LIN {X -0.238,Y -550.331,Z 626.317,A 0.000,B 0.000,C 90.000,E1 273.037} C_DIS
LIN {X 0.107,Y -549.893,Z 626.307,A 0.000,B 0.000,C 90.000,E1 271.318} C_DIS
LIN {X -0.168,Y -549.462,Z 626.300,A 0.000,B 0.000,C 90.000,E1 269.943} C_DIS
LIN {X 0.147,Y -548.699,Z 626.290,A 0.000,B 0.000,C 90.000,E1 268.224} C_DIS
LIN {X -0.112,Y -548.146,Z 626.282,A 0.000,B 0.000,C 90.000,E1 266.846} C_DIS
LIN {X 0.223,Y -547.232,Z 626.273,A 0.000,B 0.000,C 90.000,E1 265.122} C_DIS
LIN {X 0.038,Y -546.174,Z 626.264,A 0.000,B 0.000,C 90.000,E1 263.451} C_DIS
LIN {X 0.258,Y -545.222,Z 626.257,A 0.000,B 0.000,C 90.000,E1 262.299} C_DIS
LIN {X -0.006,Y -544.035,Z 626.251,A 0.000,B 0.000,C 90.000,E1 261.197} C_DIS
LIN {X -0.034,Y -541.933,Z 626.240,A 0.000,B 0.000,C 90.000,E1 259.218} C_DIS
LIN {X -0.086,Y -540.451,Z 626.231,A 0.000,B 0.000,C 90.000,E1 257.521} C_DIS
LIN {X -0.049,Y -539.015,Z 626.221,A 0.000,B 0.000,C 90.000,E1 255.811} C_DIS
LIN {X -0.172,Y -538.017,Z 626.215,A 0.000,B 0.000,C 90.000,E1 254.685} C_DIS
LIN {X -0.058,Y -536.158,Z 626.205,A 0.000,B 0.000,C 90.000,E1 252.960} C_DIS
LIN {X 0.159,Y -534.446,Z 626.196,A 0.000,B 0.000,C 90.000,E1 251.221} C_DIS
LIN {X 0.082,Y -533.521,Z 626.191,A 0.000,B 0.000,C 90.000,E1 250.369} C_DIS
LIN {X -0.105,Y -531.542,Z 626.183,A 0.000,B 0.000,C 90.000,E1 248.954} C_DIS
LIN {X -0.024,Y -529.805,Z 626.177,A 0.000,B 0.000,C 90.000,E1 247.794} C_DIS
LIN {X 0.227,Y -527.864,Z 626.170,A 0.000,B 0.000,C 90.000,E1 246.613} C_DIS
LIN {X -0.036,Y -525.751,Z 626.164,A 0.000,B 0.000,C 90.000,E1 245.485} C_DIS
LIN {X 0.208,Y -524.043,Z 626.159,A 0.000,B 0.000,C 90.000,E1 244.588} C_DIS
LIN {X 0.265,Y -520.906,Z 626.151,A 0.000,B 0.000,C 90.000,E1 243.127} C_DIS
LIN {X 0.039,Y -517.691,Z 626.143,A 0.000,B 0.000,C 90.000,E1 241.691} C_DIS
LIN {X -0.152,Y -515.079,Z 626.136,A 0.000,B 0.000,C 90.000,E1 240.539} C_DIS
LIN {X 0.122,Y -512.327,Z 626.130,A 0.000,B 0.000,C 90.000,E1 239.331} C_DIS
LIN {X -0.008,Y -508.763,Z 626.122,A 0.000,B 0.000,C 90.000,E1 237.867} C_DIS
LIN {X -0.258,Y -505.789,Z 626.115,A 0.000,B 0.000,C 90.000,E1 236.707} C_DIS
LIN {X 0.036,Y -501.976,Z 626.107,A 0.000,B 0.000,C 90.000,E1 235.182} C_DIS
LIN {X -0.030,Y -498.809,Z 626.100,A 0.000,B 0.000,C 90.000,E1 233.989} C_DIS
LIN {X 0.287,Y -492.539,Z 626.087,A 0.000,B 0.000,C 90.000,E1 231.537} C_DIS
LIN {X -0.012,Y -489.480,Z 626.080,A 0.000,B 0.000,C 90.000,E1 230.356} C_DIS
LIN {X -0.065,Y -484.980,Z 626.070,A 0.000,B 0.000,C 90.000,E1 228.528} C_DIS
LIN {X 0.105,Y -480.442,Z 626.059,A 0.000,B 0.000,C 90.000,E1 226.662} C_DIS
LIN {X -0.071,Y -475.104,Z 626.047,A 0.000,B 0.000,C 90.000,E1 224.514} C_DIS
LIN {X -0.037,Y -470.081,Z 626.035,A 0.000,B 0.000,C 90.000,E1 222.324} C_DIS
LIN {X 0.031,Y -466.677,Z 626.026,A 0.000,B 0.000,C 90.000,E1 220.744} C_DIS
LIN {X 0.018,Y -463.990,Z 626.019,A 0.000,B 0.000,C 90.000,E1 219.483} C_DIS
LIN {X -0.178,Y -459.941,Z 626.009,A 0.000,B 0.000,C 90.000,E1 217.604} C_DIS
LIN {X -0.097,Y -455.501,Z 625.996,A 0.000,B 0.000,C 90.000,E1 215.358} C_DIS
LIN {X 0.072,Y -451.396,Z 625.984,A 0.000,B 0.000,C 90.000,E1 213.086} C_DIS
LIN {X -0.118,Y -447.220,Z 625.971,A 0.000,B 0.000,C 90.000,E1 210.846} C_DIS
LIN {X 0.057,Y -443.799,Z 625.961,A 0.000,B 0.000,C 90.000,E1 208.871} C_DIS
LIN {X -0.104,Y -440.885,Z 625.951,A 0.000,B 0.000,C 90.000,E1 207.257} C_DIS
LIN {X 0.073,Y -438.014,Z 625.942,A 0.000,B 0.000,C 90.000,E1 205.591} C_DIS
LIN {X -0.168,Y -434.449,Z 625.931,A 0.000,B 0.000,C 90.000,E1 203.643} C_DIS
LIN {X -0.077,Y -431.571,Z 625.922,A 0.000,B 0.000,C 90.000,E1 201.972} C_DIS
LIN {X 0.163,Y -428.191,Z 625.911,A 0.000,B 0.000,C 90.000,E1 199.939} C_DIS
LIN {X 0.030,Y -424.888,Z 625.900,A 0.000,B 0.000,C 90.000,E1 197.946} C_DIS
LIN {X 0.039,Y -422.294,Z 625.890,A 0.000,B 0.000,C 90.000,E1 196.260} C_DIS
LIN {X -0.129,Y -419.795,Z 625.881,A 0.000,B 0.000,C 90.000,E1 194.592} C_DIS
LIN {X -0.101,Y -417.703,Z 625.873,A 0.000,B 0.000,C 90.000,E1 193.231} C_DIS
LIN {X -0.107,Y -414.553,Z 625.862,A 0.000,B 0.000,C 90.000,E1 191.186} C_DIS
LIN {X -0.217,Y -411.248,Z 625.849,A 0.000,B 0.000,C 90.000,E1 188.803} C_DIS
LIN {X -0.120,Y -408.829,Z 625.839,A 0.000,B 0.000,C 90.000,E1 187.068} C_DIS
LIN {X -0.135,Y -405.186,Z 625.824,A 0.000,B 0.000,C 90.000,E1 184.302} C_DIS
LIN {X 0.067,Y -402.053,Z 625.808,A 0.000,B 0.000,C 90.000,E1 181.489} C_DIS
LIN {X -0.006,Y -398.738,Z 625.787,A 0.000,B 0.000,C 90.000,E1 177.650} C_DIS
LIN {X -0.094,Y -396.919,Z 625.767,A 0.000,B 0.000,C 90.000,E1 174.147} C_DIS
LIN {X -0.033,Y -396.196,Z 625.752,A 0.000,B 0.000,C 90.000,E1 171.319} C_DIS
LIN {X -0.170,Y -395.877,Z 625.738,A 0.000,B 0.000,C 90.000,E1 168.870} C_DIS
LIN {X 0.157,Y -395.965,Z 625.724,A 0.000,B 0.000,C 90.000,E1 166.353} C_DIS
LIN {X -0.121,Y -396.213,Z 625.715,A 0.000,B 0.000,C 90.000,E1 164.629} C_DIS
LIN {X -0.190,Y -396.744,Z 625.699,A 0.000,B 0.000,C 90.000,E1 161.819} C_DIS
LIN {X -0.077,Y -397.316,Z 625.685,A 0.000,B 0.000,C 90.000,E1 159.337} C_DIS
LIN {X -0.046,Y -398.043,Z 625.672,A 0.000,B 0.000,C 90.000,E1 156.869} C_DIS
LIN {X 0.029,Y -398.608,Z 625.662,A 0.000,B 0.000,C 90.000,E1 155.101} C_DIS
LIN {X -0.131,Y -399.372,Z 625.648,A 0.000,B 0.000,C 90.000,E1 152.666} C_DIS
LIN {X -0.206,Y -399.932,Z 625.638,A 0.000,B 0.000,C 90.000,E1 150.923} C_DIS
LIN {X 0.118,Y -400.462,Z 625.629,A 0.000,B 0.000,C 90.000,E1 149.125} C_DIS
LIN {X 0.113,Y -400.964,Z 625.619,A 0.000,B 0.000,C 90.000,E1 147.375} C_DIS
LIN {X -0.112,Y -401.664,Z 625.607,A 0.000,B 0.000,C 90.000,E1 145.308} C_DIS
LIN {X -0.097,Y -402.475,Z 625.596,A 0.000,B 0.000,C 90.000,E1 143.210} C_DIS
LIN {X -0.033,Y -403.162,Z 625.586,A 0.000,B 0.000,C 90.000,E1 141.457} C_DIS
LIN {X -0.085,Y -403.660,Z 625.578,A 0.000,B 0.000,C 90.000,E1 140.070} C_DIS
LIN {X 0.077,Y -404.308,Z 625.567,A 0.000,B 0.000,C 90.000,E1 137.957} C_DIS
LIN {X 0.096,Y -404.746,Z 625.557,A 0.000,B 0.000,C 90.000,E1 136.215} C_DIS
LIN {X 0.245,Y -405.355,Z 625.545,A 0.000,B 0.000,C 90.000,E1 134.109} C_DIS
LIN {X -0.011,Y -406.207,Z 625.532,A 0.000,B 0.000,C 90.000,E1 131.714} C_DIS
LIN {X -0.107,Y -407.674,Z 625.516,A 0.000,B 0.000,C 90.000,E1 128.955} C_DIS
LIN {X 0.039,Y -408.028,Z 625.514,A 0.000,B 0.000,C 90.000,E1 128.588} C_DIS
LIN {X -0.085,Y -410.807,Z 625.509,A 0.000,B 0.000,C 90.000,E1 127.569} C_DIS
LIN {X 0.149,Y -415.361,Z 625.500,A 0.000,B 0.000,C 90.000,E1 126.011} C_DIS
LIN {X -0.048,Y -416.301,Z 625.500,A 0.000,B 0.000,C 90.000,E1 125.931} C_DIS
LIN {X -0.097,Y -420.149,Z 625.498,A 0.000,B 0.000,C 90.000,E1 125.598} C_DIS
LIN {X -0.058,Y -424.196,Z 625.496,A 0.000,B 0.000,C 90.000,E1 125.311} C_DIS
LIN {X 0.097,Y -437.399,Z 625.492,A 0.000,B 0.000,C 90.000,E1 124.532} C_DIS
LIN {X -0.193,Y -449.189,Z 625.488,A 0.000,B 0.000,C 90.000,E1 123.913} C_DIS
LIN {X -0.123,Y -457.391,Z 625.486,A 0.000,B 0.000,C 90.000,E1 123.420} C_DIS
LIN {X 0.004,Y -466.760,Z 625.482,A 0.000,B 0.000,C 90.000,E1 122.832} C_DIS
LIN {X 0.064,Y -476.279,Z 625.479,A 0.000,B 0.000,C 90.000,E1 122.212} C_DIS
LIN {X 0.108,Y -484.143,Z 625.476,A 0.000,B 0.000,C 90.000,E1 121.671} C_DIS
LIN {X 0.109,Y -493.504,Z 625.472,A 0.000,B 0.000,C 90.000,E1 121.003} C_DIS
LIN {X -0.146,Y -501.117,Z 625.469,A 0.000,B 0.000,C 90.000,E1 120.463} C_DIS
LIN {X 0.061,Y -508.352,Z 625.466,A 0.000,B 0.000,C 90.000,E1 119.873} C_DIS
LIN {X 0.094,Y -518.447,Z 625.461,A 0.000,B 0.000,C 90.000,E1 119.027} C_DIS
LIN {X 0.070,Y -525.476,Z 625.458,A 0.000,B 0.000,C 90.000,E1 118.409} C_DIS
LIN {X 0.108,Y -529.640,Z 625.456,A 0.000,B 0.000,C 90.000,E1 118.025} C_DIS
LIN {X 0.020,Y -535.127,Z 625.453,A 0.000,B 0.000,C 90.000,E1 117.513} C_DIS
LIN {X -0.133,Y -538.731,Z 625.451,A 0.000,B 0.000,C 90.000,E1 117.180} C_DIS
LIN {X -0.136,Y -543.458,Z 625.448,A 0.000,B 0.000,C 90.000,E1 116.668} C_DIS
LIN {X -0.003,Y -548.137,Z 625.445,A 0.000,B 0.000,C 90.000,E1 116.104} C_DIS
LIN {X 0.010,Y -552.376,Z 625.442,A 0.000,B 0.000,C 90.000,E1 115.540} C_DIS
LIN {X -0.054,Y -557.008,Z 625.438,A 0.000,B 0.000,C 90.000,E1 114.847} C_DIS
LIN {X 0.052,Y -561.642,Z 625.434,A 0.000,B 0.000,C 90.000,E1 114.027} C_DIS
LIN {X -0.030,Y -565.882,Z 625.429,A 0.000,B 0.000,C 90.000,E1 113.206} C_DIS
LIN {X -0.070,Y -569.554,Z 625.424,A 0.000,B 0.000,C 90.000,E1 112.386} C_DIS
LIN {X 0.060,Y -574.179,Z 625.418,A 0.000,B 0.000,C 90.000,E1 111.280} C_DIS
LIN {X 0.056,Y -578.279,Z 625.412,A 0.000,B 0.000,C 90.000,E1 110.194} C_DIS
LIN {X -0.078,Y -581.071,Z 625.408,A 0.000,B 0.000,C 90.000,E1 109.396} C_DIS
LIN {X -0.190,Y -583.566,Z 625.403,A 0.000,B 0.000,C 90.000,E1 108.598} C_DIS
LIN {X -0.063,Y -586.495,Z 625.397,A 0.000,B 0.000,C 90.000,E1 107.511} C_DIS
LIN {X -0.157,Y -587.866,Z 625.394,A 0.000,B 0.000,C 90.000,E1 106.985} C_DIS
LIN {X -0.284,Y -591.159,Z 625.387,A 0.000,B 0.000,C 90.000,E1 105.662} C_DIS
LIN {X -0.266,Y -596.613,Z 625.375,A 0.000,B 0.000,C 90.000,E1 103.536} C_DIS
LIN {X -0.265,Y -599.399,Z 625.369,A 0.000,B 0.000,C 90.000,E1 102.479} C_DIS
LIN {X -0.197,Y -603.575,Z 625.360,A 0.000,B 0.000,C 90.000,E1 100.894} C_DIS
LIN {X 0.107,Y -607.006,Z 625.353,A 0.000,B 0.000,C 90.000,E1 99.557} C_DIS
LIN {X -0.135,Y -610.174,Z 625.346,A 0.000,B 0.000,C 90.000,E1 98.276} C_DIS
LIN {X 0.193,Y -614.271,Z 625.336,A 0.000,B 0.000,C 90.000,E1 96.429} C_DIS
LIN {X 0.229,Y -616.302,Z 625.330,A 0.000,B 0.000,C 90.000,E1 95.391} C_DIS
LIN {X -0.073,Y -618.525,Z 625.323,A 0.000,B 0.000,C 90.000,E1 94.131} C_DIS
LIN {X -0.292,Y -620.574,Z 625.316,A 0.000,B 0.000,C 90.000,E1 92.865} C_DIS
LIN {X 0.051,Y -621.668,Z 625.312,A 0.000,B 0.000,C 90.000,E1 92.064} C_DIS
LIN {X 0.136,Y -622.808,Z 625.306,A 0.000,B 0.000,C 90.000,E1 91.031} C_DIS
LIN {X 0.221,Y -623.787,Z 625.300,A 0.000,B 0.000,C 90.000,E1 90.000} C_DIS
LIN {X -0.018,Y -624.268,Z 625.296,A 0.000,B 0.000,C 90.000,E1 89.255} C_DIS
LIN {X 0.081,Y -624.675,Z 625.290,A 0.000,B 0.000,C 90.000,E1 88.224} C_DIS
LIN {X -0.134,Y -624.734,Z 625.286,A 0.000,B 0.000,C 90.000,E1 87.478} C_DIS
LIN {X -0.295,Y -624.585,Z 625.279,A 0.000,B 0.000,C 90.000,E1 86.216} C_DIS
LIN {X 0.118,Y -624.262,Z 625.275,A 0.000,B 0.000,C 90.000,E1 85.412} C_DIS
LIN {X -0.013,Y -623.489,Z 625.268,A 0.000,B 0.000,C 90.000,E1 84.147} C_DIS
LIN {X -0.087,Y -622.462,Z 625.260,A 0.000,B 0.000,C 90.000,E1 82.875} C_DIS
LIN {X -0.326,Y -621.689,Z 625.256,A 0.000,B 0.000,C 90.000,E1 82.129} C_DIS
LIN {X -0.110,Y -620.289,Z 625.250,A 0.000,B 0.000,C 90.000,E1 81.084} C_DIS
LIN {X 0.091,Y -618.680,Z 625.245,A 0.000,B 0.000,C 90.000,E1 80.038} C_DIS
LIN {X 0.264,Y -616.968,Z 625.239,A 0.000,B 0.000,C 90.000,E1 78.993} C_DIS
LIN {X 0.293,Y -614.515,Z 625.232,A 0.000,B 0.000,C 90.000,E1 77.701} C_DIS
LIN {X 0.285,Y -611.826,Z 625.225,A 0.000,B 0.000,C 90.000,E1 76.408} C_DIS
LIN {X -0.366,Y -608.884,Z 625.217,A 0.000,B 0.000,C 90.000,E1 75.172} C_DIS
LIN {X -0.156,Y -605.788,Z 625.210,A 0.000,B 0.000,C 90.000,E1 73.850} C_DIS
LIN {X 0.109,Y -603.138,Z 625.204,A 0.000,B 0.000,C 90.000,E1 72.779} C_DIS
LIN {X 0.034,Y -600.930,Z 625.200,A 0.000,B 0.000,C 90.000,E1 72.000} C_DIS
LIN {X -0.066,Y -598.465,Z 625.196,A 0.000,B 0.000,C 90.000,E1 71.221} C_DIS
LIN {X 0.104,Y -596.734,Z 625.193,A 0.000,B 0.000,C 90.000,E1 70.678} C_DIS
LIN {X 0.154,Y -593.854,Z 625.188,A 0.000,B 0.000,C 90.000,E1 69.880} C_DIS
LIN {X 0.178,Y -590.751,Z 625.184,A 0.000,B 0.000,C 90.000,E1 69.082} C_DIS
LIN {X 0.052,Y -586.222,Z 625.178,A 0.000,B 0.000,C 90.000,E1 68.028} C_DIS
LIN {X -0.002,Y -582.655,Z 625.174,A 0.000,B 0.000,C 90.000,E1 67.230} C_DIS
LIN {X -0.104,Y -578.747,Z 625.169,A 0.000,B 0.000,C 90.000,E1 66.433} C_DIS
LIN {X 0.057,Y -575.327,Z 625.165,A 0.000,B 0.000,C 90.000,E1 65.741} C_DIS
LIN {X 0.186,Y -571.594,Z 625.162,A 0.000,B 0.000,C 90.000,E1 65.049} C_DIS
LIN {X -0.320,Y -566.558,Z 625.157,A 0.000,B 0.000,C 90.000,E1 64.280} C_DIS
LIN {X 0.075,Y -562.924,Z 625.154,A 0.000,B 0.000,C 90.000,E1 63.691} C_DIS
LIN {X 0.191,Y -558.910,Z 625.151,A 0.000,B 0.000,C 90.000,E1 63.127} C_DIS
LIN {X -0.219,Y -554.473,Z 625.148,A 0.000,B 0.000,C 90.000,E1 62.615} C_DIS
LIN {X -0.336,Y -549.951,Z 625.145,A 0.000,B 0.000,C 90.000,E1 62.103} C_DIS
LIN {X 0.070,Y -543.792,Z 625.141,A 0.000,B 0.000,C 90.000,E1 61.435} C_DIS
LIN {X -0.135,Y -539.718,Z 625.139,A 0.000,B 0.000,C 90.000,E1 61.101} C_DIS
LIN {X -0.158,Y -534.269,Z 625.137,A 0.000,B 0.000,C 90.000,E1 60.667} C_DIS
LIN {X -0.155,Y -528.322,Z 625.135,A 0.000,B 0.000,C 90.000,E1 60.255} C_DIS
LIN {X -0.188,Y -521.929,Z 625.133,A 0.000,B 0.000,C 90.000,E1 59.871} C_DIS
LIN {X 0.181,Y -515.321,Z 625.130,A 0.000,B 0.000,C 90.000,E1 59.459} C_DIS
LIN {X -0.259,Y -507.004,Z 625.128,A 0.000,B 0.000,C 90.000,E1 59.076} C_DIS
LIN {X -0.021,Y -486.670,Z 625.122,A 0.000,B 0.000,C 90.000,E1 58.043} C_DIS
LIN {X -0.163,Y -464.653,Z 625.116,A 0.000,B 0.000,C 90.000,E1 56.962} C_DIS
LIN {X 0.071,Y -444.690,Z 625.111,A 0.000,B 0.000,C 90.000,E1 55.881} C_DIS
LIN {X -0.024,Y -442.057,Z 625.110,A 0.000,B 0.000,C 90.000,E1 55.754} C_DIS
LIN {X -0.066,Y -442.035,Z 625.110,A 0.000,B 0.000,C 90.000,E1 55.754} C_DIS
LIN {X 0.119,Y -433.238,Z 625.088,A 0.000,B 0.000,C 90.000,E1 51.743} C_DIS
LIN {X 0.026,Y -431.392,Z 625.082,A 0.000,B 0.000,C 90.000,E1 50.759} C_DIS
LIN {X 0.229,Y -426.619,Z 625.071,A 0.000,B 0.000,C 90.000,E1 48.771} C_DIS
LIN {X -0.030,Y -427.146,Z 625.065,A 0.000,B 0.000,C 90.000,E1 47.757} C_DIS
LIN {X 0.093,Y -427.920,Z 625.054,A 0.000,B 0.000,C 90.000,E1 45.729} C_DIS
LIN {X 0.056,Y -428.728,Z 625.039,A 0.000,B 0.000,C 90.000,E1 43.056} C_DIS
LIN {X 0.166,Y -429.719,Z 625.026,A 0.000,B 0.000,C 90.000,E1 40.701} C_DIS
LIN {X -0.221,Y -430.687,Z 625.015,A 0.000,B 0.000,C 90.000,E1 38.749} C_DIS
LIN {X -0.174,Y -431.480,Z 625.006,A 0.000,B 0.000,C 90.000,E1 37.076} C_DIS
LIN {X -0.023,Y -432.094,Z 624.997,A 0.000,B 0.000,C 90.000,E1 35.391} C_DIS
LIN {X -0.114,Y -432.517,Z 624.991,A 0.000,B 0.000,C 90.000,E1 34.405} C_DIS
LIN {X -0.197,Y -433.009,Z 624.984,A 0.000,B 0.000,C 90.000,E1 33.086} C_DIS
LIN {X 0.100,Y -433.543,Z 624.974,A 0.000,B 0.000,C 90.000,E1 31.386} C_DIS
LIN {X 0.013,Y -434.468,Z 624.960,A 0.000,B 0.000,C 90.000,E1 28.743} C_DIS
LIN {X 0.075,Y -435.055,Z 624.951,A 0.000,B 0.000,C 90.000,E1 27.078} C_DIS
LIN {X -0.061,Y -435.631,Z 624.943,A 0.000,B 0.000,C 90.000,E1 25.771} C_DIS
LIN {X 0.060,Y -436.391,Z 624.932,A 0.000,B 0.000,C 90.000,E1 23.770} C_DIS
LIN {X -0.200,Y -437.132,Z 624.923,A 0.000,B 0.000,C 90.000,E1 22.153} C_DIS
LIN {X -0.046,Y -438.014,Z 624.914,A 0.000,B 0.000,C 90.000,E1 20.482} C_DIS
LIN {X 0.075,Y -438.944,Z 624.903,A 0.000,B 0.000,C 90.000,E1 18.489} C_DIS
LIN {X 0.187,Y -440.341,Z 624.888,A 0.000,B 0.000,C 90.000,E1 15.843} C_DIS
LIN {X 0.109,Y -441.545,Z 624.877,A 0.000,B 0.000,C 90.000,E1 13.883} C_DIS
LIN {X -0.168,Y -443.357,Z 624.863,A 0.000,B 0.000,C 90.000,E1 11.299} C_DIS
LIN {X -0.021,Y -445.814,Z 624.846,A 0.000,B 0.000,C 90.000,E1 8.341} C_DIS
LIN {X -0.208,Y -447.982,Z 624.834,A 0.000,B 0.000,C 90.000,E1 6.087} C_DIS
LIN {X -0.128,Y -449.992,Z 624.823,A 0.000,B 0.000,C 90.000,E1 4.131} C_DIS
LIN {X 0.029,Y -453.394,Z 624.807,A 0.000,B 0.000,C 90.000,E1 1.203} C_DIS
LIN {X 0.171,Y -457.509,Z 624.790,A 0.000,B 0.000,C 90.000,E1 358.167} C_DIS
LIN {X 0.174,Y -460.969,Z 624.778,A 0.000,B 0.000,C 90.000,E1 355.931} C_DIS
LIN {X -0.102,Y -463.613,Z 624.769,A 0.000,B 0.000,C 90.000,E1 354.375} C_DIS
LIN {X -0.057,Y -466.888,Z 624.758,A 0.000,B 0.000,C 90.000,E1 352.470} C_DIS
LIN {X 0.130,Y -470.097,Z 624.748,A 0.000,B 0.000,C 90.000,E1 350.557} C_DIS
LIN {X -0.086,Y -473.191,Z 624.737,A 0.000,B 0.000,C 90.000,E1 348.701} C_DIS
LIN {X 0.104,Y -475.917,Z 624.729,A 0.000,B 0.000,C 90.000,E1 347.117} C_DIS
LIN {X 0.155,Y -479.754,Z 624.716,A 0.000,B 0.000,C 90.000,E1 344.936} C_DIS
LIN {X 0.103,Y -483.850,Z 624.704,A 0.000,B 0.000,C 90.000,E1 342.779} C_DIS
LIN {X -0.162,Y -487.442,Z 624.694,A 0.000,B 0.000,C 90.000,E1 340.967} C_DIS
LIN {X 0.275,Y -490.987,Z 624.684,A 0.000,B 0.000,C 90.000,E1 339.082} C_DIS
LIN {X -0.221,Y -493.252,Z 624.677,A 0.000,B 0.000,C 90.000,E1 337.922} C_DIS
LIN {X 0.146,Y -495.356,Z 624.671,A 0.000,B 0.000,C 90.000,E1 336.666} C_DIS
LIN {X -0.104,Y -497.338,Z 624.664,A 0.000,B 0.000,C 90.000,E1 335.485} C_DIS
LIN {X -0.065,Y -499.650,Z 624.655,A 0.000,B 0.000,C 90.000,E1 333.973} C_DIS
LIN {X -0.213,Y -501.895,Z 624.647,A 0.000,B 0.000,C 90.000,E1 332.487} C_DIS
LIN {X -0.014,Y -504.556,Z 624.637,A 0.000,B 0.000,C 90.000,E1 330.667} C_DIS
LIN {X -0.005,Y -511.885,Z 624.614,A 0.000,B 0.000,C 90.000,E1 326.501} C_DIS
LIN {X 0.167,Y -514.083,Z 624.609,A 0.000,B 0.000,C 90.000,E1 325.595} C_DIS
LIN {X 0.014,Y -515.681,Z 624.606,A 0.000,B 0.000,C 90.000,E1 325.022} C_DIS
LIN {X 0.297,Y -517.558,Z 624.602,A 0.000,B 0.000,C 90.000,E1 324.402} C_DIS
LIN {X 0.157,Y -519.468,Z 624.600,A 0.000,B 0.000,C 90.000,E1 323.989} C_DIS
LIN {X 0.099,Y -521.279,Z 624.598,A 0.000,B 0.000,C 90.000,E1 323.703} C_DIS
LIN {X 0.048,Y -522.984,Z 624.597,A 0.000,B 0.000,C 90.000,E1 323.417} C_DIS
LIN {X 0.140,Y -526.185,Z 624.594,A 0.000,B 0.000,C 90.000,E1 322.970} C_DIS
LIN {X 0.049,Y -529.455,Z 624.593,A 0.000,B 0.000,C 90.000,E1 322.637} C_DIS
LIN {X 0.168,Y -532.347,Z 624.591,A 0.000,B 0.000,C 90.000,E1 322.351} C_DIS
LIN {X 0.075,Y -545.594,Z 624.585,A 0.000,B 0.000,C 90.000,E1 321.295} C_DIS
LIN {X 0.128,Y -558.508,Z 624.579,A 0.000,B 0.000,C 90.000,E1 320.231} C_DIS
LIN {X -0.046,Y -574.231,Z 624.572,A 0.000,B 0.000,C 90.000,E1 318.976} C_DIS
LIN {X 0.275,Y -582.640,Z 624.568,A 0.000,B 0.000,C 90.000,E1 318.243} C_DIS
LIN {X 0.185,Y -593.339,Z 624.563,A 0.000,B 0.000,C 90.000,E1 317.310} C_DIS
LIN {X 0.125,Y -598.440,Z 624.560,A 0.000,B 0.000,C 90.000,E1 316.863} C_DIS
LIN {X -0.229,Y -602.243,Z 624.558,A 0.000,B 0.000,C 90.000,E1 316.539} C_DIS
LIN {X -0.297,Y -607.186,Z 624.556,A 0.000,B 0.000,C 90.000,E1 316.053} C_DIS
LIN {X 0.364,Y -610.598,Z 624.554,A 0.000,B 0.000,C 90.000,E1 315.648} C_DIS
LIN {X -0.014,Y -615.083,Z 624.551,A 0.000,B 0.000,C 90.000,E1 315.202} C_DIS
LIN {X -0.263,Y -618.536,Z 624.549,A 0.000,B 0.000,C 90.000,E1 314.838} C_DIS
LIN {X -0.205,Y -623.987,Z 624.545,A 0.000,B 0.000,C 90.000,E1 314.190} C_DIS
LIN {X -0.100,Y -629.099,Z 624.542,A 0.000,B 0.000,C 90.000,E1 313.542} C_DIS
LIN {X -0.020,Y -636.856,Z 624.536,A 0.000,B 0.000,C 90.000,E1 312.528} C_DIS
LIN {X 0.084,Y -644.394,Z 624.531,A 0.000,B 0.000,C 90.000,E1 311.515} C_DIS
LIN {X -0.073,Y -651.474,Z 624.525,A 0.000,B 0.000,C 90.000,E1 310.539} C_DIS
LIN {X -0.178,Y -655.474,Z 624.522,A 0.000,B 0.000,C 90.000,E1 309.930} C_DIS
LIN {X -0.186,Y -658.454,Z 624.519,A 0.000,B 0.000,C 90.000,E1 309.439} C_DIS
LIN {X 0.247,Y -661.263,Z 624.516,A 0.000,B 0.000,C 90.000,E1 308.910} C_DIS
LIN {X -0.234,Y -663.809,Z 624.514,A 0.000,B 0.000,C 90.000,E1 308.463} C_DIS
LIN {X 0.300,Y -668.476,Z 624.508,A 0.000,B 0.000,C 90.000,E1 307.443} C_DIS
LIN {X -0.149,Y -670.643,Z 624.505,A 0.000,B 0.000,C 90.000,E1 306.996} C_DIS
LIN {X 0.080,Y -673.593,Z 624.501,A 0.000,B 0.000,C 90.000,E1 306.251} C_DIS
LIN {X -0.341,Y -675.378,Z 624.499,A 0.000,B 0.000,C 90.000,E1 305.804} C_DIS
LIN {X 0.104,Y -679.585,Z 624.492,A 0.000,B 0.000,C 90.000,E1 304.565} C_DIS
LIN {X 0.060,Y -683.525,Z 624.485,A 0.000,B 0.000,C 90.000,E1 303.372} C_DIS
LIN {X -0.306,Y -687.285,Z 624.479,A 0.000,B 0.000,C 90.000,E1 302.212} C_DIS
LIN {X -0.255,Y -690.104,Z 624.474,A 0.000,B 0.000,C 90.000,E1 301.258} C_DIS
LIN {X 0.058,Y -693.535,Z 624.467,A 0.000,B 0.000,C 90.000,E1 300.050} C_DIS
LIN {X -0.173,Y -696.119,Z 624.462,A 0.000,B 0.000,C 90.000,E1 299.127} C_DIS
LIN {X -0.445,Y -699.128,Z 624.455,A 0.000,B 0.000,C 90.000,E1 297.975} C_DIS
LIN {X -0.261,Y -700.742,Z 624.451,A 0.000,B 0.000,C 90.000,E1 297.257} C_DIS
LIN {X 0.285,Y -701.657,Z 624.449,A 0.000,B 0.000,C 90.000,E1 296.744} C_DIS
LIN {X -0.102,Y -702.433,Z 624.446,A 0.000,B 0.000,C 90.000,E1 296.309} C_DIS
LIN {X -0.173,Y -702.726,Z 624.444,A 0.000,B 0.000,C 90.000,E1 295.848} C_DIS
LIN {X 0.107,Y -702.720,Z 624.442,A 0.000,B 0.000,C 90.000,E1 295.591} C_DIS
LIN {X -0.268,Y -701.663,Z 624.440,A 0.000,B 0.000,C 90.000,E1 295.155} C_DIS
LIN {X 0.010,Y -700.925,Z 624.438,A 0.000,B 0.000,C 90.000,E1 294.899} C_DIS
LIN {X 0.148,Y -700.176,Z 624.438,A 0.000,B 0.000,C 90.000,E1 294.771} C_DIS
LIN {X -0.116,Y -696.397,Z 624.435,A 0.000,B 0.000,C 90.000,E1 294.335} C_DIS
LIN {X 0.138,Y -695.258,Z 624.435,A 0.000,B 0.000,C 90.000,E1 294.207} C_DIS
LIN {X 0.304,Y -693.387,Z 624.434,A 0.000,B 0.000,C 90.000,E1 294.079} C_DIS
LIN {X -0.243,Y -684.169,Z 624.432,A 0.000,B 0.000,C 90.000,E1 293.770} C_DIS
LIN {X -0.099,Y -681.487,Z 624.432,A 0.000,B 0.000,C 90.000,E1 293.695} C_DIS
LIN {X 0.025,Y -673.801,Z 624.431,A 0.000,B 0.000,C 90.000,E1 293.567} C_DIS
LIN {X 0.153,Y -665.018,Z 624.430,A 0.000,B 0.000,C 90.000,E1 293.462} C_DIS
LIN {X 0.290,Y -651.279,Z 624.429,A 0.000,B 0.000,C 90.000,E1 293.259} C_DIS
LIN {X -0.153,Y -641.294,Z 624.428,A 0.000,B 0.000,C 90.000,E1 293.131} C_DIS
LIN {X 0.176,Y -631.407,Z 624.427,A 0.000,B 0.000,C 90.000,E1 292.898} C_DIS
LIN {X 0.292,Y -621.654,Z 624.426,A 0.000,B 0.000,C 90.000,E1 292.642} C_DIS
LIN {X 0.022,Y -598.024,Z 624.422,A 0.000,B 0.000,C 90.000,E1 291.972} C_DIS
LIN {X 0.123,Y -578.916,Z 624.419,A 0.000,B 0.000,C 90.000,E1 291.354} C_DIS
LIN {X 0.306,Y -570.092,Z 624.417,A 0.000,B 0.000,C 90.000,E1 291.099} C_DIS
LIN {X 0.130,Y -565.522,Z 624.417,A 0.000,B 0.000,C 90.000,E1 290.972} C_DIS
LIN {X -0.006,Y -559.879,Z 624.415,A 0.000,B 0.000,C 90.000,E1 290.737} C_DIS
LIN {X -0.017,Y -558.911,Z 624.415,A 0.000,B 0.000,C 90.000,E1 290.663} C_DIS
LIN {X 0.267,Y -557.330,Z 624.414,A 0.000,B 0.000,C 90.000,E1 290.482} C_DIS
LIN {X 0.228,Y -557.309,Z 624.414,A 0.000,B 0.000,C 90.000,E1 290.482} C_DIS
LIN {X 0.188,Y -556.544,Z 624.413,A 0.000,B 0.000,C 90.000,E1 290.248} C_DIS
LIN {X -0.156,Y -556.281,Z 624.410,A 0.000,B 0.000,C 90.000,E1 289.866} C_DIS
LIN {X 0.113,Y -556.400,Z 624.404,A 0.000,B 0.000,C 90.000,E1 288.725} C_DIS
LIN {X -0.139,Y -556.375,Z 624.398,A 0.000,B 0.000,C 90.000,E1 287.638} C_DIS
LIN {X 0.136,Y -556.091,Z 624.392,A 0.000,B 0.000,C 90.000,E1 286.496} C_DIS
LIN {X -0.284,Y -555.757,Z 624.386,A 0.000,B 0.000,C 90.000,E1 285.426} C_DIS
LIN {X -0.197,Y -554.770,Z 624.375,A 0.000,B 0.000,C 90.000,E1 283.467} C_DIS
LIN {X 0.146,Y -553.817,Z 624.364,A 0.000,B 0.000,C 90.000,E1 281.478} C_DIS
LIN {X -0.297,Y -552.973,Z 624.355,A 0.000,B 0.000,C 90.000,E1 279.849} C_DIS
LIN {X 0.216,Y -552.386,Z 624.347,A 0.000,B 0.000,C 90.000,E1 278.398} C_DIS
LIN {X 0.204,Y -551.631,Z 624.338,A 0.000,B 0.000,C 90.000,E1 276.720} C_DIS
LIN {X 0.256,Y -550.782,Z 624.325,A 0.000,B 0.000,C 90.000,E1 274.473} C_DIS
LIN {X 0.040,Y -550.422,Z 624.317,A 0.000,B 0.000,C 90.000,E1 273.094} C_DIS
LIN {X -0.109,Y -549.910,Z 624.306,A 0.000,B 0.000,C 90.000,E1 271.146} C_DIS
LIN {X 0.167,Y -549.427,Z 624.299,A 0.000,B 0.000,C 90.000,E1 269.714} C_DIS
LIN {X -0.119,Y -548.833,Z 624.291,A 0.000,B 0.000,C 90.000,E1 268.339} C_DIS
LIN {X 0.220,Y -548.160,Z 624.281,A 0.000,B 0.000,C 90.000,E1 266.617} C_DIS
LIN {X 0.003,Y -547.234,Z 624.272,A 0.000,B 0.000,C 90.000,E1 264.951} C_DIS
LIN {X -0.186,Y -546.146,Z 624.263,A 0.000,B 0.000,C 90.000,E1 263.280} C_DIS
LIN {X 0.013,Y -545.428,Z 624.258,A 0.000,B 0.000,C 90.000,E1 262.413} C_DIS
LIN {X 0.294,Y -544.291,Z 624.252,A 0.000,B 0.000,C 90.000,E1 261.254} C_DIS
LIN {X 0.173,Y -542.170,Z 624.241,A 0.000,B 0.000,C 90.000,E1 259.285} C_DIS
LIN {X 0.188,Y -540.430,Z 624.230,A 0.000,B 0.000,C 90.000,E1 257.297} C_DIS
LIN {X 0.143,Y -539.248,Z 624.222,A 0.000,B 0.000,C 90.000,E1 255.880} C_DIS
LIN {X 0.015,Y -538.216,Z 624.215,A 0.000,B 0.000,C 90.000,E1 254.755} C_DIS
LIN {X 0.073,Y -536.690,Z 624.207,A 0.000,B 0.000,C 90.000,E1 253.323} C_DIS
LIN {X -0.002,Y -534.647,Z 624.196,A 0.000,B 0.000,C 90.000,E1 251.329} C_DIS
LIN {X -0.049,Y -533.365,Z 624.190,A 0.000,B 0.000,C 90.000,E1 250.188} C_DIS
LIN {X 0.061,Y -531.780,Z 624.184,A 0.000,B 0.000,C 90.000,E1 249.028} C_DIS
LIN {X -0.152,Y -530.037,Z 624.177,A 0.000,B 0.000,C 90.000,E1 247.901} C_DIS
LIN {X -0.280,Y -528.592,Z 624.172,A 0.000,B 0.000,C 90.000,E1 247.050} C_DIS
LIN {X 0.339,Y -526.007,Z 624.164,A 0.000,B 0.000,C 90.000,E1 245.537} C_DIS
LIN {X 0.051,Y -523.661,Z 624.158,A 0.000,B 0.000,C 90.000,E1 244.409} C_DIS
LIN {X 0.096,Y -520.491,Z 624.150,A 0.000,B 0.000,C 90.000,E1 242.948} C_DIS
LIN {X 0.189,Y -517.927,Z 624.143,A 0.000,B 0.000,C 90.000,E1 241.769} C_DIS
LIN {X -0.091,Y -514.614,Z 624.135,A 0.000,B 0.000,C 90.000,E1 240.333} C_DIS
LIN {X -0.171,Y -512.560,Z 624.130,A 0.000,B 0.000,C 90.000,E1 239.459} C_DIS
LIN {X -0.292,Y -508.992,Z 624.122,A 0.000,B 0.000,C 90.000,E1 237.995} C_DIS
LIN {X -0.111,Y -506.029,Z 624.115,A 0.000,B 0.000,C 90.000,E1 236.786} C_DIS
LIN {X 0.183,Y -502.166,Z 624.107,A 0.000,B 0.000,C 90.000,E1 235.261} C_DIS
LIN {X 0.116,Y -499.004,Z 624.101,A 0.000,B 0.000,C 90.000,E1 234.069} C_DIS
LIN {X 0.045,Y -492.745,Z 624.087,A 0.000,B 0.000,C 90.000,E1 231.662} C_DIS
LIN {X 0.126,Y -488.131,Z 624.077,A 0.000,B 0.000,C 90.000,E1 229.828} C_DIS
LIN {X -0.099,Y -484.350,Z 624.068,A 0.000,B 0.000,C 90.000,E1 228.324} C_DIS
LIN {X 0.049,Y -479.802,Z 624.058,A 0.000,B 0.000,C 90.000,E1 226.458} C_DIS
LIN {X 0.288,Y -473.753,Z 624.044,A 0.000,B 0.000,C 90.000,E1 223.947} C_DIS
LIN {X 0.278,Y -468.828,Z 624.032,A 0.000,B 0.000,C 90.000,E1 221.757} C_DIS
LIN {X 0.006,Y -465.436,Z 624.023,A 0.000,B 0.000,C 90.000,E1 220.216} C_DIS
LIN {X -0.026,Y -462.697,Z 624.016,A 0.000,B 0.000,C 90.000,E1 218.955} C_DIS
LIN {X -0.020,Y -460.057,Z 624.009,A 0.000,B 0.000,C 90.000,E1 217.684} C_DIS
LIN {X 0.067,Y -455.608,Z 623.997,A 0.000,B 0.000,C 90.000,E1 215.438} C_DIS
LIN {X -0.137,Y -451.497,Z 623.984,A 0.000,B 0.000,C 90.000,E1 213.214} C_DIS
LIN {X 0.058,Y -447.308,Z 623.972,A 0.000,B 0.000,C 90.000,E1 210.924} C_DIS
LIN {X 0.239,Y -443.873,Z 623.961,A 0.000,B 0.000,C 90.000,E1 208.949} C_DIS
LIN {X 0.242,Y -441.570,Z 623.954,A 0.000,B 0.000,C 90.000,E1 207.641} C_DIS
LIN {X -0.128,Y -438.084,Z 623.943,A 0.000,B 0.000,C 90.000,E1 205.720} C_DIS
LIN {X -0.039,Y -436.310,Z 623.937,A 0.000,B 0.000,C 90.000,E1 204.719} C_DIS
LIN {X 0.073,Y -432.252,Z 623.924,A 0.000,B 0.000,C 90.000,E1 202.386} C_DIS
LIN {X -0.022,Y -428.306,Z 623.911,A 0.000,B 0.000,C 90.000,E1 200.066} C_DIS
LIN {X -0.016,Y -424.984,Z 623.900,A 0.000,B 0.000,C 90.000,E1 198.055} C_DIS
LIN {X 0.051,Y -421.859,Z 623.889,A 0.000,B 0.000,C 90.000,E1 196.024} C_DIS
LIN {X -0.123,Y -419.398,Z 623.880,A 0.000,B 0.000,C 90.000,E1 194.356} C_DIS
LIN {X -0.050,Y -416.790,Z 623.870,A 0.000,B 0.000,C 90.000,E1 192.647} C_DIS
LIN {X 0.013,Y -412.745,Z 623.855,A 0.000,B 0.000,C 90.000,E1 189.905} C_DIS
LIN {X 0.163,Y -410.908,Z 623.847,A 0.000,B 0.000,C 90.000,E1 188.511} C_DIS
LIN {X -0.159,Y -408.484,Z 623.838,A 0.000,B 0.000,C 90.000,E1 186.834} C_DIS
LIN {X -0.195,Y -405.352,Z 623.824,A 0.000,B 0.000,C 90.000,E1 184.416} C_DIS
LIN {X 0.011,Y -402.203,Z 623.809,A 0.000,B 0.000,C 90.000,E1 181.604} C_DIS
LIN {X -0.055,Y -398.882,Z 623.788,A 0.000,B 0.000,C 90.000,E1 177.764} C_DIS
LIN {X -0.134,Y -397.042,Z 623.768,A 0.000,B 0.000,C 90.000,E1 174.261} C_DIS
LIN {X -0.064,Y -396.277,Z 623.752,A 0.000,B 0.000,C 90.000,E1 171.432} C_DIS
LIN {X 0.152,Y -396.000,Z 623.741,A 0.000,B 0.000,C 90.000,E1 169.285} C_DIS
LIN {X 0.089,Y -396.033,Z 623.727,A 0.000,B 0.000,C 90.000,E1 166.825} C_DIS
LIN {X 0.193,Y -396.270,Z 623.717,A 0.000,B 0.000,C 90.000,E1 165.046} C_DIS
LIN {X 0.128,Y -396.771,Z 623.701,A 0.000,B 0.000,C 90.000,E1 162.236} C_DIS
LIN {X -0.123,Y -397.334,Z 623.688,A 0.000,B 0.000,C 90.000,E1 159.806} C_DIS
LIN {X 0.075,Y -397.953,Z 623.676,A 0.000,B 0.000,C 90.000,E1 157.667} C_DIS
LIN {X 0.217,Y -398.662,Z 623.664,A 0.000,B 0.000,C 90.000,E1 155.537} C_DIS
LIN {X 0.008,Y -399.307,Z 623.653,A 0.000,B 0.000,C 90.000,E1 153.461} C_DIS
LIN {X -0.194,Y -400.021,Z 623.641,A 0.000,B 0.000,C 90.000,E1 151.385} C_DIS
LIN {X 0.020,Y -400.680,Z 623.629,A 0.000,B 0.000,C 90.000,E1 149.253} C_DIS
LIN {X 0.022,Y -401.153,Z 623.620,A 0.000,B 0.000,C 90.000,E1 147.502} C_DIS
LIN {X 0.136,Y -401.872,Z 623.608,A 0.000,B 0.000,C 90.000,E1 145.388} C_DIS
LIN {X -0.045,Y -402.772,Z 623.594,A 0.000,B 0.000,C 90.000,E1 142.970} C_DIS
LIN {X -0.220,Y -403.453,Z 623.585,A 0.000,B 0.000,C 90.000,E1 141.251} C_DIS
LIN {X -0.011,Y -403.918,Z 623.577,A 0.000,B 0.000,C 90.000,E1 139.828} C_DIS
LIN {X 0.032,Y -404.443,Z 623.567,A 0.000,B 0.000,C 90.000,E1 138.081} C_DIS
LIN {X 0.186,Y -404.949,Z 623.556,A 0.000,B 0.000,C 90.000,E1 135.972} C_DIS
LIN {X -0.232,Y -405.536,Z 623.544,A 0.000,B 0.000,C 90.000,E1 133.947} C_DIS
LIN {X -0.051,Y -406.224,Z 623.532,A 0.000,B 0.000,C 90.000,E1 131.838} C_DIS
LIN {X 0.050,Y -407.780,Z 623.515,A 0.000,B 0.000,C 90.000,E1 128.705} C_DIS
LIN {X -0.034,Y -408.091,Z 623.514,A 0.000,B 0.000,C 90.000,E1 128.543} C_DIS
LIN {X -0.068,Y -415.579,Z 623.500,A 0.000,B 0.000,C 90.000,E1 125.964} C_DIS
LIN {X -0.111,Y -416.155,Z 623.498,A 0.000,B 0.000,C 90.000,E1 125.724} C_DIS
LIN {X -0.150,Y -416.180,Z 623.498,A 0.000,B 0.000,C 90.000,E1 125.724} C_DIS
LIN {X 0.001,Y -418.680,Z 623.497,A 0.000,B 0.000,C 90.000,E1 125.471} C_DIS
LIN {X -0.024,Y -422.992,Z 623.495,A 0.000,B 0.000,C 90.000,E1 125.152} C_DIS
LIN {X 0.071,Y -438.645,Z 623.490,A 0.000,B 0.000,C 90.000,E1 124.246} C_DIS
LIN {X 0.052,Y -447.247,Z 623.488,A 0.000,B 0.000,C 90.000,E1 123.785} C_DIS
LIN {X 0.259,Y -458.835,Z 623.484,A 0.000,B 0.000,C 90.000,E1 123.086} C_DIS
LIN {X 0.137,Y -466.714,Z 623.481,A 0.000,B 0.000,C 90.000,E1 122.625} C_DIS
LIN {X 0.249,Y -473.009,Z 623.479,A 0.000,B 0.000,C 90.000,E1 122.212} C_DIS
LIN {X 0.120,Y -482.589,Z 623.476,A 0.000,B 0.000,C 90.000,E1 121.592} C_DIS
LIN {X 0.249,Y -491.998,Z 623.472,A 0.000,B 0.000,C 90.000,E1 120.924} C_DIS
LIN {X 0.318,Y -502.760,Z 623.468,A 0.000,B 0.000,C 90.000,E1 120.129} C_DIS
LIN {X -0.109,Y -510.099,Z 623.464,A 0.000,B 0.000,C 90.000,E1 119.589} C_DIS
LIN {X 0.226,Y -518.915,Z 623.460,A 0.000,B 0.000,C 90.000,E1 118.821} C_DIS
LIN {X -0.083,Y -526.049,Z 623.457,A 0.000,B 0.000,C 90.000,E1 118.231} C_DIS
LIN {X -0.214,Y -534.029,Z 623.453,A 0.000,B 0.000,C 90.000,E1 117.513} C_DIS
LIN {X -0.244,Y -538.080,Z 623.451,A 0.000,B 0.000,C 90.000,E1 117.129} C_DIS
LIN {X 0.007,Y -543.115,Z 623.448,A 0.000,B 0.000,C 90.000,E1 116.565} C_DIS
LIN {X 0.264,Y -548.006,Z 623.445,A 0.000,B 0.000,C 90.000,E1 115.976} C_DIS
LIN {X -0.220,Y -552.388,Z 623.441,A 0.000,B 0.000,C 90.000,E1 115.463} C_DIS
LIN {X -0.287,Y -557.088,Z 623.438,A 0.000,B 0.000,C 90.000,E1 114.771} C_DIS
LIN {X 0.199,Y -561.213,Z 623.434,A 0.000,B 0.000,C 90.000,E1 114.027} C_DIS
LIN {X 0.215,Y -564.909,Z 623.430,A 0.000,B 0.000,C 90.000,E1 113.334} C_DIS
LIN {X 0.260,Y -568.132,Z 623.426,A 0.000,B 0.000,C 90.000,E1 112.642} C_DIS
LIN {X -0.152,Y -572.906,Z 623.420,A 0.000,B 0.000,C 90.000,E1 111.589} C_DIS
LIN {X -0.175,Y -575.162,Z 623.417,A 0.000,B 0.000,C 90.000,E1 111.046} C_DIS
LIN {X -0.342,Y -578.272,Z 623.412,A 0.000,B 0.000,C 90.000,E1 110.248} C_DIS
LIN {X 0.067,Y -581.125,Z 623.408,A 0.000,B 0.000,C 90.000,E1 109.396} C_DIS
LIN {X -0.045,Y -583.692,Z 623.403,A 0.000,B 0.000,C 90.000,E1 108.598} C_DIS
LIN {X 0.240,Y -585.989,Z 623.399,A 0.000,B 0.000,C 90.000,E1 107.764} C_DIS
LIN {X -0.006,Y -588.081,Z 623.394,A 0.000,B 0.000,C 90.000,E1 106.985} C_DIS
LIN {X -0.128,Y -591.429,Z 623.387,A 0.000,B 0.000,C 90.000,E1 105.662} C_DIS
LIN {X -0.101,Y -596.905,Z 623.375,A 0.000,B 0.000,C 90.000,E1 103.536} C_DIS
LIN {X -0.096,Y -599.753,Z 623.369,A 0.000,B 0.000,C 90.000,E1 102.479} C_DIS
LIN {X -0.018,Y -603.952,Z 623.361,A 0.000,B 0.000,C 90.000,E1 100.894} C_DIS
LIN {X 0.294,Y -607.457,Z 623.353,A 0.000,B 0.000,C 90.000,E1 99.557} C_DIS
LIN {X 0.060,Y -610.682,Z 623.346,A 0.000,B 0.000,C 90.000,E1 98.276} C_DIS
LIN {X -0.209,Y -614.846,Z 623.336,A 0.000,B 0.000,C 90.000,E1 96.486} C_DIS
LIN {X 0.126,Y -617.404,Z 623.329,A 0.000,B 0.000,C 90.000,E1 95.163} C_DIS
LIN {X -0.109,Y -619.615,Z 623.322,A 0.000,B 0.000,C 90.000,E1 93.898} C_DIS
LIN {X 0.271,Y -621.645,Z 623.315,A 0.000,B 0.000,C 90.000,E1 92.579} C_DIS
LIN {X 0.007,Y -622.693,Z 623.310,A 0.000,B 0.000,C 90.000,E1 91.835} C_DIS
LIN {X -0.184,Y -624.049,Z 623.303,A 0.000,B 0.000,C 90.000,E1 90.573} C_DIS
LIN {X 0.204,Y -624.701,Z 623.299,A 0.000,B 0.000,C 90.000,E1 89.771} C_DIS
LIN {X -0.027,Y -625.137,Z 623.295,A 0.000,B 0.000,C 90.000,E1 89.026} C_DIS
LIN {X 0.103,Y -625.438,Z 623.289,A 0.000,B 0.000,C 90.000,E1 87.993} C_DIS
LIN {X -0.126,Y -625.479,Z 623.285,A 0.000,B 0.000,C 90.000,E1 87.249} C_DIS
LIN {X 0.010,Y -625.305,Z 623.279,A 0.000,B 0.000,C 90.000,E1 86.216} C_DIS
LIN {X 0.190,Y -624.799,Z 623.273,A 0.000,B 0.000,C 90.000,E1 85.179} C_DIS
LIN {X -0.310,Y -624.159,Z 623.268,A 0.000,B 0.000,C 90.000,E1 84.204} C_DIS
LIN {X -0.140,Y -623.340,Z 623.262,A 0.000,B 0.000,C 90.000,E1 83.166} C_DIS
LIN {X -0.290,Y -622.577,Z 623.258,A 0.000,B 0.000,C 90.000,E1 82.413} C_DIS
LIN {X 0.173,Y -621.656,Z 623.253,A 0.000,B 0.000,C 90.000,E1 81.602} C_DIS
LIN {X 0.065,Y -619.727,Z 623.246,A 0.000,B 0.000,C 90.000,E1 80.330} C_DIS
LIN {X 0.021,Y -617.529,Z 623.239,A 0.000,B 0.000,C 90.000,E1 79.050} C_DIS
LIN {X 0.063,Y -615.042,Z 623.232,A 0.000,B 0.000,C 90.000,E1 77.757} C_DIS
LIN {X 0.067,Y -612.297,Z 623.225,A 0.000,B 0.000,C 90.000,E1 76.464} C_DIS
LIN {X 0.269,Y -609.923,Z 623.219,A 0.000,B 0.000,C 90.000,E1 75.408} C_DIS
LIN {X -0.258,Y -606.834,Z 623.212,A 0.000,B 0.000,C 90.000,E1 74.157} C_DIS
LIN {X 0.017,Y -604.160,Z 623.206,A 0.000,B 0.000,C 90.000,E1 73.087} C_DIS
LIN {X -0.050,Y -601.977,Z 623.202,A 0.000,B 0.000,C 90.000,E1 72.308} C_DIS
LIN {X 0.049,Y -599.586,Z 623.197,A 0.000,B 0.000,C 90.000,E1 71.511} C_DIS
LIN {X -0.064,Y -596.934,Z 623.193,A 0.000,B 0.000,C 90.000,E1 70.732} C_DIS
LIN {X -0.008,Y -593.975,Z 623.189,A 0.000,B 0.000,C 90.000,E1 69.934} C_DIS
LIN {X 0.022,Y -590.834,Z 623.184,A 0.000,B 0.000,C 90.000,E1 69.135} C_DIS
LIN {X -0.318,Y -586.199,Z 623.178,A 0.000,B 0.000,C 90.000,E1 68.103} C_DIS
LIN {X 0.320,Y -581.886,Z 623.173,A 0.000,B 0.000,C 90.000,E1 67.102} C_DIS
LIN {X -0.249,Y -578.595,Z 623.169,A 0.000,B 0.000,C 90.000,E1 66.485} C_DIS
LIN {X -0.087,Y -575.085,Z 623.166,A 0.000,B 0.000,C 90.000,E1 65.793} C_DIS
LIN {X 0.212,Y -571.325,Z 623.162,A 0.000,B 0.000,C 90.000,E1 65.101} C_DIS
LIN {X -0.206,Y -567.062,Z 623.158,A 0.000,B 0.000,C 90.000,E1 64.460} C_DIS
LIN {X -0.148,Y -562.387,Z 623.154,A 0.000,B 0.000,C 90.000,E1 63.768} C_DIS
LIN {X 0.087,Y -558.399,Z 623.151,A 0.000,B 0.000,C 90.000,E1 63.204} C_DIS
LIN {X 0.195,Y -552.948,Z 623.148,A 0.000,B 0.000,C 90.000,E1 62.538} C_DIS
LIN {X 0.329,Y -548.512,Z 623.145,A 0.000,B 0.000,C 90.000,E1 62.025} C_DIS
LIN {X 0.206,Y -543.084,Z 623.142,A 0.000,B 0.000,C 90.000,E1 61.513} C_DIS
LIN {X 0.232,Y -537.616,Z 623.139,A 0.000,B 0.000,C 90.000,E1 61.051} C_DIS
LIN {X 0.084,Y -533.072,Z 623.137,A 0.000,B 0.000,C 90.000,E1 60.717} C_DIS
LIN {X 0.072,Y -526.315,Z 623.135,A 0.000,B 0.000,C 90.000,E1 60.284} C_DIS
LIN {X 0.257,Y -519.618,Z 623.133,A 0.000,B 0.000,C 90.000,E1 59.871} C_DIS
LIN {X 0.121,Y -514.739,Z 623.131,A 0.000,B 0.000,C 90.000,E1 59.616} C_DIS
LIN {X 0.012,Y -507.939,Z 623.129,A 0.000,B 0.000,C 90.000,E1 59.282} C_DIS
LIN {X -0.087,Y -489.323,Z 623.124,A 0.000,B 0.000,C 90.000,E1 58.377} C_DIS
LIN {X -0.062,Y -477.377,Z 623.121,A 0.000,B 0.000,C 90.000,E1 57.788} C_DIS
LIN {X 0.239,Y -467.388,Z 623.118,A 0.000,B 0.000,C 90.000,E1 57.248} C_DIS
LIN {X -0.009,Y -445.520,Z 623.112,A 0.000,B 0.000,C 90.000,E1 56.135} C_DIS
LIN {X -0.145,Y -442.747,Z 623.111,A 0.000,B 0.000,C 90.000,E1 56.008} C_DIS
LIN {X -0.188,Y -442.642,Z 623.111,A 0.000,B 0.000,C 90.000,E1 56.008} C_DIS
LIN {X 0.165,Y -433.712,Z 623.089,A 0.000,B 0.000,C 90.000,E1 51.984} C_DIS
LIN {X 0.011,Y -431.860,Z 623.083,A 0.000,B 0.000,C 90.000,E1 51.009} C_DIS
LIN {X -0.002,Y -431.175,Z 623.082,A 0.000,B 0.000,C 90.000,E1 50.678} C_DIS
LIN {X -0.060,Y -427.035,Z 623.072,A 0.000,B 0.000,C 90.000,E1 48.976} C_DIS
LIN {X -0.055,Y -427.702,Z 623.065,A 0.000,B 0.000,C 90.000,E1 47.676} C_DIS
LIN {X 0.162,Y -428.377,Z 623.056,A 0.000,B 0.000,C 90.000,E1 45.972} C_DIS
LIN {X 0.143,Y -429.281,Z 623.041,A 0.000,B 0.000,C 90.000,E1 43.299} C_DIS
LIN {X -0.055,Y -430.281,Z 623.028,A 0.000,B 0.000,C 90.000,E1 40.987} C_DIS
LIN {X -0.077,Y -431.080,Z 623.018,A 0.000,B 0.000,C 90.000,E1 39.322} C_DIS
LIN {X -0.025,Y -431.879,Z 623.009,A 0.000,B 0.000,C 90.000,E1 37.649} C_DIS
LIN {X -0.217,Y -432.558,Z 623.000,A 0.000,B 0.000,C 90.000,E1 36.011} C_DIS
LIN {X -0.053,Y -433.089,Z 622.993,A 0.000,B 0.000,C 90.000,E1 34.659} C_DIS
LIN {X -0.119,Y -433.660,Z 622.983,A 0.000,B 0.000,C 90.000,E1 33.007} C_DIS
LIN {X -0.057,Y -434.057,Z 622.976,A 0.000,B 0.000,C 90.000,E1 31.671} C_DIS
LIN {X 0.074,Y -434.789,Z 622.963,A 0.000,B 0.000,C 90.000,E1 29.333} C_DIS
LIN {X -0.042,Y -435.375,Z 622.954,A 0.000,B 0.000,C 90.000,E1 27.692} C_DIS
LIN {X 0.034,Y -436.025,Z 622.945,A 0.000,B 0.000,C 90.000,E1 26.027} C_DIS
LIN {X -0.234,Y -436.757,Z 622.934,A 0.000,B 0.000,C 90.000,E1 24.079} C_DIS
LIN {X 0.081,Y -437.466,Z 622.924,A 0.000,B 0.000,C 90.000,E1 22.386} C_DIS
LIN {X -0.081,Y -438.420,Z 622.914,A 0.000,B 0.000,C 90.000,E1 20.429} C_DIS
LIN {X -0.060,Y -439.176,Z 622.904,A 0.000,B 0.000,C 90.000,E1 18.779} C_DIS
LIN {X 0.048,Y -440.508,Z 622.890,A 0.000,B 0.000,C 90.000,E1 16.134} C_DIS
LIN {X 0.120,Y -441.886,Z 622.877,A 0.000,B 0.000,C 90.000,E1 13.828} C_DIS
LIN {X -0.144,Y -443.670,Z 622.862,A 0.000,B 0.000,C 90.000,E1 11.243} C_DIS
LIN {X 0.083,Y -446.127,Z 622.846,A 0.000,B 0.000,C 90.000,E1 8.276} C_DIS
LIN {X -0.109,Y -448.260,Z 622.833,A 0.000,B 0.000,C 90.000,E1 6.024} C_DIS
LIN {X -0.068,Y -450.248,Z 622.823,A 0.000,B 0.000,C 90.000,E1 4.073} C_DIS
LIN {X -0.071,Y -453.238,Z 622.808,A 0.000,B 0.000,C 90.000,E1 1.489} C_DIS
LIN {X -0.011,Y -457.180,Z 622.792,A 0.000,B 0.000,C 90.000,E1 358.511} C_DIS
LIN {X -0.014,Y -460.584,Z 622.779,A 0.000,B 0.000,C 90.000,E1 356.274} C_DIS
LIN {X -0.092,Y -463.723,Z 622.769,A 0.000,B 0.000,C 90.000,E1 354.375} C_DIS
LIN {X 0.159,Y -467.550,Z 622.756,A 0.000,B 0.000,C 90.000,E1 352.129} C_DIS
LIN {X 0.144,Y -470.175,Z 622.748,A 0.000,B 0.000,C 90.000,E1 350.557} C_DIS
LIN {X -0.242,Y -473.788,Z 622.735,A 0.000,B 0.000,C 90.000,E1 348.409} C_DIS
LIN {X -0.041,Y -476.505,Z 622.727,A 0.000,B 0.000,C 90.000,E1 346.825} C_DIS
LIN {X 0.174,Y -479.820,Z 622.716,A 0.000,B 0.000,C 90.000,E1 344.936} C_DIS
LIN {X 0.124,Y -483.915,Z 622.704,A 0.000,B 0.000,C 90.000,E1 342.779} C_DIS
LIN {X -0.122,Y -488.086,Z 622.693,A 0.000,B 0.000,C 90.000,E1 340.659} C_DIS
LIN {X -0.160,Y -491.052,Z 622.684,A 0.000,B 0.000,C 90.000,E1 339.135} C_DIS
LIN {X -0.195,Y -493.280,Z 622.677,A 0.000,B 0.000,C 90.000,E1 337.922} C_DIS
LIN {X 0.172,Y -495.384,Z 622.671,A 0.000,B 0.000,C 90.000,E1 336.666} C_DIS
LIN {X -0.077,Y -497.365,Z 622.664,A 0.000,B 0.000,C 90.000,E1 335.485} C_DIS
LIN {X -0.038,Y -499.678,Z 622.655,A 0.000,B 0.000,C 90.000,E1 333.973} C_DIS
LIN {X -0.186,Y -501.922,Z 622.647,A 0.000,B 0.000,C 90.000,E1 332.487} C_DIS
LIN {X 0.015,Y -504.554,Z 622.637,A 0.000,B 0.000,C 90.000,E1 330.667} C_DIS
LIN {X -0.067,Y -512.379,Z 622.612,A 0.000,B 0.000,C 90.000,E1 326.215} C_DIS
